LIN {X 0,Y 516.96,Z 356.095,A -85,B 0,C 180,E1 -5071.105,E2 -5071.105} C_VEL
LIN {X 0,Y 516.912,Z 356.1,A -85,B 0,C 180,E1 -5073.966,E2 -5073.966} C_VEL
LIN {X 0,Y 516.88,Z 356.104,A -85,B 0,C 180,E1 -5076.746,E2 -5076.746} C_VEL
LIN {X 0,Y 516.915,Z 356.098,A -85,B 0,C 180,E1 -5079.718,E2 -5079.718} C_VEL
LIN {X 0,Y 516.909,Z 356.099,A -85,B 0,C 180,E1 -5082.829,E2 -5082.829} C_VEL
LIN {X 0,Y 516.926,Z 356.097,A -85,B 0,C 180,E1 -5085.01,E2 -5085.01} C_VEL
LIN {X 0,Y 516.919,Z 356.099,A -85,B 0,C 180,E1 -5088.398,E2 -5088.398} C_VEL
LIN {X 0,Y 516.883,Z 356.103,A -85,B 0,C 180,E1 -5091.284,E2 -5091.284} C_VEL
LIN {X 0,Y 516.874,Z 356.103,A -85,B 0,C 180,E1 -5094.22,E2 -5094.22} C_VEL
LIN {X 0,Y 516.899,Z 356.103,A -85,B 0,C 180,E1 -5097.053,E2 -5097.053} C_VEL
LIN {X 0,Y 516.917,Z 356.245,A -85,B 0,C 180,E1 -5098.494,E2 -5098.494} C_VEL
LIN {X 0,Y 518.951,Z 365.114,A -85,B 0,C 180,E1 -5100.821,E2 -5100.821} C_VEL
LIN {X 0,Y 519.572,Z 369.036,A -85,B 0,C 180,E1 -5101.743,E2 -5101.743} C_VEL
LIN {X 0,Y 518.932,Z 379.362,A -85,B 0,C 180,E1 -5103.886,E2 -5103.886} C_VEL
LIN {X 0,Y 518.227,Z 395.981,A -85,B 0,C 180,E1 -5107.107,E2 -5107.107} C_VEL
LIN {X 0,Y 517.651,Z 412.713,A -85,B 0,C 180,E1 -5110.158,E2 -5110.158} C_VEL
LIN {X 0,Y 517.309,Z 428.9,A -85,B 0,C 180,E1 -5113.017,E2 -5113.017} C_VEL
LIN {X 0,Y 516.99,Z 447.206,A -85,B 0,C 180,E1 -5116.137,E2 -5116.137} C_VEL
LIN {X 0,Y 518.34,Z 458.651,A -85,B 0,C 180,E1 -5116.399,E2 -5116.399} C_VEL
LIN {X 0,Y 518.166,Z 471.053,A -85,B 0,C 180,E1 -5116.769,E2 -5116.769} C_VEL
LIN {X 0,Y 517.921,Z 483.766,A -85,B 0,C 180,E1 -5117.311,E2 -5117.311} C_VEL
LIN {X 0,Y 517.637,Z 495.546,A -85,B 0,C 180,E1 -5117.976,E2 -5117.976} C_VEL
LIN {X 0,Y 517.405,Z 506.176,A -85,B 0,C 180,E1 -5118.74,E2 -5118.74} C_VEL
LIN {X 0,Y 517.111,Z 516.148,A -85,B 0,C 180,E1 -5119.625,E2 -5119.625} C_VEL
LIN {X 0,Y 516.856,Z 525.214,A -85,B 0,C 180,E1 -5120.609,E2 -5120.609} C_VEL
LIN {X 0,Y 516.656,Z 534.061,A -85,B 0,C 180,E1 -5121.788,E2 -5121.788} C_VEL
LIN {X 0,Y 516.507,Z 541.106,A -85,B 0,C 180,E1 -5122.966,E2 -5122.966} C_VEL
LIN {X 0,Y 516.454,Z 546.751,A -85,B 0,C 180,E1 -5124.142,E2 -5124.142} C_VEL
LIN {X 0,Y 516.271,Z 551.161,A -85,B 0,C 180,E1 -5125.315,E2 -5125.315} C_VEL
LIN {X 0,Y 516.372,Z 553.512,A -85,B 0,C 180,E1 -5126.098,E2 -5126.098} C_VEL
LIN {X 0,Y 516.282,Z 555.403,A -85,B 0,C 180,E1 -5126.878,E2 -5126.878} C_VEL
LIN {X 0,Y 516.261,Z 556.824,A -85,B 0,C 180,E1 -5127.659,E2 -5127.659} C_VEL
LIN {X 0,Y 516.16,Z 558.448,A -85,B 0,C 180,E1 -5129.22,E2 -5129.22} C_VEL
LIN {X 0,Y 516.155,Z 558.67,A -85,B 0,C 180,E1 -5130,E2 -5130} C_VEL
LIN {X 0,Y 516.192,Z 557.838,A -85,B 0,C 180,E1 -5131.56,E2 -5131.56} C_VEL
LIN {X 0,Y 516.261,Z 556.835,A -85,B 0,C 180,E1 -5132.34,E2 -5132.34} C_VEL
LIN {X 0,Y 516.282,Z 555.417,A -85,B 0,C 180,E1 -5133.121,E2 -5133.121} C_VEL
LIN {X 0,Y 516.343,Z 552.441,A -85,B 0,C 180,E1 -5134.293,E2 -5134.293} C_VEL
LIN {X 0,Y 516.405,Z 548.405,A -85,B 0,C 180,E1 -5135.467,E2 -5135.467} C_VEL
LIN {X 0,Y 516.463,Z 543.024,A -85,B 0,C 180,E1 -5136.677,E2 -5136.677} C_VEL
LIN {X 0,Y 516.578,Z 536.641,A -85,B 0,C 180,E1 -5137.819,E2 -5137.819} C_VEL
LIN {X 0,Y 516.771,Z 528.471,A -85,B 0,C 180,E1 -5138.998,E2 -5138.998} C_VEL
LIN {X 0,Y 516.992,Z 520.13,A -85,B 0,C 180,E1 -5139.981,E2 -5139.981} C_VEL
LIN {X 0,Y 517.294,Z 509.933,A -85,B 0,C 180,E1 -5140.965,E2 -5140.965} C_VEL
LIN {X 0,Y 517.565,Z 498.759,A -85,B 0,C 180,E1 -5141.824,E2 -5141.824} C_VEL
LIN {X 0,Y 517.875,Z 486.984,A -85,B 0,C 180,E1 -5142.541,E2 -5142.541} C_VEL
LIN {X 0,Y 518.09,Z 475.398,A -85,B 0,C 180,E1 -5143.083,E2 -5143.083} C_VEL
LIN {X 0,Y 518.347,Z 462.076,A -85,B 0,C 180,E1 -5143.526,E2 -5143.526} C_VEL
LIN {X 0,Y 518.143,Z 456.418,A -85,B 0,C 180,E1 -5143.669,E2 -5143.669} C_VEL
LIN {X 0,Y 516.994,Z 447.607,A -85,B 0,C 180,E1 -5143.862,E2 -5143.862} C_VEL
LIN {X 0,Y 517.335,Z 430.732,A -85,B 0,C 180,E1 -5146.779,E2 -5146.779} C_VEL
LIN {X 0,Y 517.768,Z 411.104,A -85,B 0,C 180,E1 -5150.182,E2 -5150.182} C_VEL
LIN {X 0,Y 518.432,Z 392.937,A -85,B 0,C 180,E1 -5153.572,E2 -5153.572} C_VEL
LIN {X 0,Y 519.014,Z 377.127,A -85,B 0,C 180,E1 -5156.542,E2 -5156.542} C_VEL
LIN {X 0,Y 519.331,Z 367.451,A -85,B 0,C 180,E1 -5158.402,E2 -5158.402} C_VEL
LIN {X 0,Y 516.899,Z 356.101,A -85,B 0,C 180,E1 -5160.893,E2 -5160.893} C_VEL
LIN {X 0,Y 516.91,Z 356.098,A -85,B 0,C 180,E1 -5163.966,E2 -5163.966} C_VEL
LIN {X 0,Y 516.878,Z 356.103,A -85,B 0,C 180,E1 -5166.746,E2 -5166.746} C_VEL
LIN {X 0,Y 516.883,Z 356.099,A -85,B 0,C 180,E1 -5169.721,E2 -5169.721} C_VEL
LIN {X 0,Y 516.908,Z 356.095,A -85,B 0,C 180,E1 -5172.76,E2 -5172.76} C_VEL
LIN {X 0,Y 516.924,Z 356.097,A -85,B 0,C 180,E1 -5175.01,E2 -5175.01} C_VEL
LIN {X 0,Y 516.917,Z 356.099,A -85,B 0,C 180,E1 -5178.398,E2 -5178.398} C_VEL
LIN {X 0,Y 516.884,Z 356.098,A -85,B 0,C 180,E1 -5181.284,E2 -5181.284} C_VEL
LIN {X 0,Y 516.891,Z 356.098,A -85,B 0,C 180,E1 -5184.221,E2 -5184.221} C_VEL
LIN {X 0,Y 516.896,Z 356.1,A -85,B 0,C 180,E1 -5187.053,E2 -5187.053} C_VEL
LIN {X 0,Y 516.894,Z 356.098,A -85,B 0,C 180,E1 -5189.796,E2 -5189.796} C_VEL
LIN {X 0,Y 516.93,Z 356.092,A -85,B 0,C 180,E1 -5192.467,E2 -5192.467} C_VEL
LIN {X 0,Y 516.91,Z 356.098,A -85,B 0,C 180,E1 -5195.072,E2 -5195.072} C_VEL
LIN {X 0,Y 516.888,Z 356.102,A -85,B 0,C 180,E1 -5198.462,E2 -5198.462} C_VEL
LIN {X 0,Y 516.904,Z 356.095,A -85,B 0,C 180,E1 -5200.955,E2 -5200.955} C_VEL
LIN {X 0,Y 516.916,Z 356.097,A -85,B 0,C 180,E1 -5203.41,E2 -5203.41} C_VEL
LIN {X 0,Y 516.908,Z 356.096,A -85,B 0,C 180,E1 -5205.834,E2 -5205.834} C_VEL
LIN {X 0,Y 516.954,Z 356.091,A -85,B 0,C 180,E1 -5209.028,E2 -5209.028} C_VEL
LIN {X 0,Y 516.98,Z 356.088,A -85,B 0,C 180,E1 -5212.187,E2 -5212.187} C_VEL
LIN {X 0,Y 517.032,Z 356.079,A -85,B 0,C 180,E1 -5214.54,E2 -5214.54} C_VEL
LIN {X 0,Y 517.084,Z 356.074,A -85,B 0,C 180,E1 -5217.663,E2 -5217.663} C_VEL
LIN {X 0,Y 517.096,Z 356.073,A -85,B 0,C 180,E1 -5220.779,E2 -5220.779} C_VEL
LIN {X 0,Y 517.014,Z 356.083,A -85,B 0,C 180,E1 -5223.117,E2 -5223.117} C_VEL
LIN {X 0,Y 517.012,Z 356.082,A -85,B 0,C 180,E1 -5226.243,E2 -5226.243} C_VEL
LIN {X 0,Y 516.956,Z 356.09,A -85,B 0,C 180,E1 -5229.389,E2 -5229.389} C_VEL
LIN {X 0,Y 516.986,Z 356.09,A -85,B 0,C 180,E1 -5231.824,E2 -5231.824} C_VEL
LIN {X 0,Y 516.946,Z 356.094,A -85,B 0,C 180,E1 -5235.147,E2 -5235.147} C_VEL
LIN {X 0,Y 516.927,Z 356.094,A -85,B 0,C 180,E1 -5238.222,E2 -5238.222} C_VEL
LIN {X 0,Y 516.914,Z 356.096,A -85,B 0,C 180,E1 -5240.701,E2 -5240.701} C_VEL
LIN {X 0,Y 516.913,Z 356.095,A -85,B 0,C 180,E1 -5244.072,E2 -5244.072} C_VEL
LIN {X 0,Y 516.926,Z 356.094,A -85,B 0,C 180,E1 -5246.658,E2 -5246.658} C_VEL
LIN {X 0,Y 516.913,Z 356.095,A -85,B 0,C 180,E1 -5249.524,E2 -5249.524} C_VEL
LIN {X 0,Y 516.899,Z 356.097,A -85,B 0,C 180,E1 -5252.544,E2 -5252.544} C_VEL
LIN {X 0,Y 516.881,Z 356.103,A -85,B 0,C 180,E1 -5255.332,E2 -5255.332} C_VEL
LIN {X 0,Y 516.883,Z 356.097,A -85,B 0,C 180,E1 -5257.943,E2 -5257.943} C_VEL
LIN {X 0,Y 516.887,Z 356.1,A -85,B 0,C 180,E1 -5260.742,E2 -5260.742} C_VEL
LIN {X 0,Y 516.885,Z 356.098,A -85,B 0,C 180,E1 -5262.831,E2 -5262.831} C_VEL
LIN {X 0,Y 516.924,Z 356.096,A -85,B 0,C 180,E1 -5265.01,E2 -5265.01} C_VEL
LIN {X 0,Y 516.918,Z 356.096,A -85,B 0,C 180,E1 -5268.399,E2 -5268.399} C_VEL
LIN {X 0,Y 516.883,Z 356.102,A -85,B 0,C 180,E1 -5270.3,E2 -5270.3} C_VEL
LIN {X 0,Y 516.212,Z 356.183,A -85,B 0,C 180,E1 -5270.95,E2 -5270.95} C_VEL
LIN {X 0,Y 513.365,Z 356.541,A -85,B 0,C 180,E1 -5272.006,E2 -5272.006} C_VEL
LIN {X 0,Y 510.955,Z 356.843,A -85,B 0,C 180,E1 -5272.856,E2 -5272.856} C_VEL
LIN {X 0,Y 509.912,Z 356.971,A -85,B 0,C 180,E1 -5273.513,E2 -5273.513} C_VEL
LIN {X 0,Y 509.822,Z 356.98,A -85,B 0,C 180,E1 -5273.735,E2 -5273.735} C_VEL
LIN {X 0,Y 509.862,Z 356.974,A -85,B 0,C 180,E1 -5276.539,E2 -5276.539} C_VEL
LIN {X 0,Y 509.848,Z 356.973,A -85,B 0,C 180,E1 -5279.334,E2 -5279.334} C_VEL
LIN {X 0,Y 509.897,Z 356.973,A -85,B 0,C 180,E1 -5282.055,E2 -5282.055} C_VEL
LIN {X 0,Y 509.879,Z 356.972,A -85,B 0,C 180,E1 -5284.704,E2 -5284.704} C_VEL
LIN {X 0,Y 509.829,Z 356.978,A -85,B 0,C 180,E1 -5287.458,E2 -5287.458} C_VEL
LIN {X 0,Y 509.92,Z 356.966,A -85,B 0,C 180,E1 -5289.845,E2 -5289.845} C_VEL
LIN {X 0,Y 509.888,Z 356.97,A -85,B 0,C 180,E1 -5293.175,E2 -5293.175} C_VEL
LIN {X 0,Y 509.867,Z 356.976,A -85,B 0,C 180,E1 -5295.634,E2 -5295.634} C_VEL
LIN {X 0,Y 509.917,Z 356.969,A -85,B 0,C 180,E1 -5298.875,E2 -5298.875} C_VEL
LIN {X 0,Y 509.955,Z 356.967,A -85,B 0,C 180,E1 -5302.079,E2 -5302.079} C_VEL
LIN {X 0,Y 509.984,Z 356.958,A -85,B 0,C 180,E1 -5304.464,E2 -5304.464} C_VEL
LIN {X 0,Y 510.059,Z 356.949,A -85,B 0,C 180,E1 -5307.631,E2 -5307.631} C_VEL
LIN {X 0,Y 510.067,Z 356.949,A -85,B 0,C 180,E1 -5310.79,E2 -5310.79} C_VEL
LIN {X 0,Y 509.957,Z 356.96,A -85,B 0,C 180,E1 -5313.16,E2 -5313.16} C_VEL
LIN {X 0,Y 509.958,Z 356.961,A -85,B 0,C 180,E1 -5316.33,E2 -5316.33} C_VEL
LIN {X 0,Y 509.919,Z 356.969,A -85,B 0,C 180,E1 -5318.72,E2 -5318.72} C_VEL
LIN {X 0,Y 509.908,Z 356.971,A -85,B 0,C 180,E1 -5321.932,E2 -5321.932} C_VEL
LIN {X 0,Y 509.898,Z 356.971,A -85,B 0,C 180,E1 -5325.242,E2 -5325.242} C_VEL
LIN {X 0,Y 509.886,Z 356.97,A -85,B 0,C 180,E1 -5327.999,E2 -5327.999} C_VEL
LIN {X 0,Y 509.854,Z 356.975,A -85,B 0,C 180,E1 -5331.002,E2 -5331.002} C_VEL
LIN {X 0,Y 509.827,Z 356.981,A -85,B 0,C 180,E1 -5333.564,E2 -5333.564} C_VEL
LIN {X 0,Y 509.916,Z 356.966,A -85,B 0,C 180,E1 -5336.379,E2 -5336.379} C_VEL
LIN {X 0,Y 509.881,Z 356.975,A -85,B 0,C 180,E1 -5338.844,E2 -5338.844} C_VEL
LIN {X 0,Y 509.825,Z 356.979,A -85,B 0,C 180,E1 -5341.59,E2 -5341.59} C_VEL
LIN {X 0,Y 509.851,Z 356.974,A -85,B 0,C 180,E1 -5344.414,E2 -5344.414} C_VEL
LIN {X 0,Y 509.82,Z 356.982,A -85,B 0,C 180,E1 -5347.341,E2 -5347.341} C_VEL
LIN {X 0,Y 509.842,Z 356.979,A -85,B 0,C 180,E1 -5350.382,E2 -5350.382} C_VEL
LIN {X 0,Y 509.843,Z 356.976,A -85,B 0,C 180,E1 -5353.064,E2 -5353.064} C_VEL
LIN {X 0,Y 509.826,Z 356.979,A -85,B 0,C 180,E1 -5355.793,E2 -5355.793} C_VEL
LIN {X 0,Y 509.859,Z 356.975,A -85,B 0,C 180,E1 -5358.575,E2 -5358.575} C_VEL
LIN {X 0,Y 509.855,Z 356.976,A -85,B 0,C 180,E1 -5361.786,E2 -5361.786} C_VEL
LIN {X 0,Y 509.847,Z 356.975,A -85,B 0,C 180,E1 -5364.623,E2 -5364.623} C_VEL
LIN {X 0,Y 509.865,Z 356.975,A -85,B 0,C 180,E1 -5367.481,E2 -5367.481} C_VEL
LIN {X 0,Y 509.955,Z 357.04,A -85,B 0,C 180,E1 -5369.925,E2 -5369.925} C_VEL
LIN {X 0,Y 509.798,Z 363.427,A -85,B 0,C 180,E1 -5372.939,E2 -5372.939} C_VEL
LIN {X 0,Y 509.694,Z 369.046,A -85,B 0,C 180,E1 -5375.565,E2 -5375.565} C_VEL
LIN {X 0,Y 509.588,Z 374.525,A -85,B 0,C 180,E1 -5378.138,E2 -5378.138} C_VEL
LIN {X 0,Y 509.5,Z 379.893,A -85,B 0,C 180,E1 -5380.667,E2 -5380.667} C_VEL
LIN {X 0,Y 509.406,Z 385.315,A -85,B 0,C 180,E1 -5383.158,E2 -5383.158} C_VEL
LIN {X 0,Y 509.378,Z 390.782,A -85,B 0,C 180,E1 -5385.62,E2 -5385.62} C_VEL
LIN {X 0,Y 509.278,Z 398.149,A -85,B 0,C 180,E1 -5388.86,E2 -5388.86} C_VEL
LIN {X 0,Y 509.269,Z 404.776,A -85,B 0,C 180,E1 -5391.718,E2 -5391.718} C_VEL
LIN {X 0,Y 510.102,Z 412.51,A -85,B 0,C 180,E1 -5392.031,E2 -5392.031} C_VEL
LIN {X 0,Y 509.994,Z 422.565,A -85,B 0,C 180,E1 -5392.577,E2 -5392.577} C_VEL
LIN {X 0,Y 509.86,Z 430.431,A -85,B 0,C 180,E1 -5393.156,E2 -5393.156} C_VEL
LIN {X 0,Y 509.631,Z 437.924,A -85,B 0,C 180,E1 -5393.865,E2 -5393.865} C_VEL
LIN {X 0,Y 509.591,Z 444.394,A -85,B 0,C 180,E1 -5394.658,E2 -5394.658} C_VEL
LIN {X 0,Y 509.512,Z 450.616,A -85,B 0,C 180,E1 -5395.649,E2 -5395.649} C_VEL
LIN {X 0,Y 509.513,Z 454.382,A -85,B 0,C 180,E1 -5396.441,E2 -5396.441} C_VEL
LIN {X 0,Y 509.254,Z 458.441,A -85,B 0,C 180,E1 -5397.627,E2 -5397.627} C_VEL
LIN {X 0,Y 509.191,Z 460.209,A -85,B 0,C 180,E1 -5398.418,E2 -5398.418} C_VEL
LIN {X 0,Y 509.173,Z 461.279,A -85,B 0,C 180,E1 -5399.209,E2 -5399.209} C_VEL
LIN {X 0,Y 509.173,Z 461.683,A -85,B 0,C 180,E1 -5400,E2 -5400} C_VEL
LIN {X 0,Y 509.179,Z 461.428,A -85,B 0,C 180,E1 -5400.791,E2 -5400.791} C_VEL
LIN {X 0,Y 509.202,Z 460.51,A -85,B 0,C 180,E1 -5401.582,E2 -5401.582} C_VEL
LIN {X 0,Y 509.381,Z 457.808,A -85,B 0,C 180,E1 -5402.768,E2 -5402.768} C_VEL
LIN {X 0,Y 509.51,Z 455.083,A -85,B 0,C 180,E1 -5403.559,E2 -5403.559} C_VEL
LIN {X 0,Y 509.532,Z 450.473,A -85,B 0,C 180,E1 -5404.549,E2 -5404.549} C_VEL
LIN {X 0,Y 509.641,Z 445.61,A -85,B 0,C 180,E1 -5405.341,E2 -5405.341} C_VEL
LIN {X 0,Y 509.731,Z 439.426,A -85,B 0,C 180,E1 -5406.134,E2 -5406.134} C_VEL
LIN {X 0,Y 509.963,Z 432.423,A -85,B 0,C 180,E1 -5406.838,E2 -5406.838} C_VEL
LIN {X 0,Y 510.044,Z 424.158,A -85,B 0,C 180,E1 -5407.482,E2 -5407.482} C_VEL
LIN {X 0,Y 510.246,Z 414.949,A -85,B 0,C 180,E1 -5408.017,E2 -5408.017} C_VEL
LIN {X 0,Y 509.775,Z 408.095,A -85,B 0,C 180,E1 -5408.323,E2 -5408.323} C_VEL
LIN {X 0,Y 509.349,Z 405.631,A -85,B 0,C 180,E1 -5408.43,E2 -5408.43} C_VEL
LIN {X 0,Y 509.46,Z 398.545,A -85,B 0,C 180,E1 -5411.636,E2 -5411.636} C_VEL
LIN {X 0,Y 509.576,Z 390.773,A -85,B 0,C 180,E1 -5415.192,E2 -5415.192} C_VEL
LIN {X 0,Y 509.663,Z 383.695,A -85,B 0,C 180,E1 -5418.491,E2 -5418.491} C_VEL
LIN {X 0,Y 509.766,Z 378.33,A -85,B 0,C 180,E1 -5421.005,E2 -5421.005} C_VEL
LIN {X 0,Y 509.885,Z 372.925,A -85,B 0,C 180,E1 -5423.561,E2 -5423.561} C_VEL
LIN {X 0,Y 510.067,Z 367.004,A -85,B 0,C 180,E1 -5426.413,E2 -5426.413} C_VEL
LIN {X 0,Y 510.222,Z 360.055,A -85,B 0,C 180,E1 -5429.728,E2 -5429.728} C_VEL
LIN {X 0,Y 509.89,Z 356.976,A -85,B 0,C 180,E1 -5431.287,E2 -5431.287} C_VEL
LIN {X 0,Y 509.851,Z 356.979,A -85,B 0,C 180,E1 -5434.414,E2 -5434.414} C_VEL
LIN {X 0,Y 509.82,Z 356.982,A -85,B 0,C 180,E1 -5437.341,E2 -5437.341} C_VEL
LIN {X 0,Y 509.866,Z 356.977,A -85,B 0,C 180,E1 -5440.38,E2 -5440.38} C_VEL
LIN {X 0,Y 509.844,Z 356.98,A -85,B 0,C 180,E1 -5443.064,E2 -5443.064} C_VEL
LIN {X 0,Y 509.834,Z 356.98,A -85,B 0,C 180,E1 -5445.792,E2 -5445.792} C_VEL
LIN {X 0,Y 509.861,Z 356.978,A -85,B 0,C 180,E1 -5448.575,E2 -5448.575} C_VEL
LIN {X 0,Y 509.853,Z 356.979,A -85,B 0,C 180,E1 -5451.786,E2 -5451.786} C_VEL
LIN {X 0,Y 509.833,Z 356.982,A -85,B 0,C 180,E1 -5454.622,E2 -5454.622} C_VEL
LIN {X 0,Y 509.867,Z 356.979,A -85,B 0,C 180,E1 -5457.481,E2 -5457.481} C_VEL
LIN {X 0,Y 509.874,Z 357.195,A -85,B 0,C 180,E1 -5458.065,E2 -5458.065} C_VEL
LIN {X 0,Y 511.829,Z 365.557,A -85,B 0,C 180,E1 -5460.375,E2 -5460.375} C_VEL
LIN {X 0,Y 512.613,Z 369.385,A -85,B 0,C 180,E1 -5461.336,E2 -5461.336} C_VEL
LIN {X 0,Y 512.479,Z 375.336,A -85,B 0,C 180,E1 -5462.651,E2 -5462.651} C_VEL
LIN {X 0,Y 511.447,Z 391.148,A -85,B 0,C 180,E1 -5465.87,E2 -5465.87} C_VEL
LIN {X 0,Y 510.911,Z 404.42,A -85,B 0,C 180,E1 -5468.409,E2 -5468.409} C_VEL
LIN {X 0,Y 510.48,Z 420.361,A -85,B 0,C 180,E1 -5471.331,E2 -5471.331} C_VEL
LIN {X 0,Y 510.135,Z 434.33,A -85,B 0,C 180,E1 -5473.801,E2 -5473.801} C_VEL
LIN {X 0,Y 509.904,Z 446.963,A -85,B 0,C 180,E1 -5476.004,E2 -5476.004} C_VEL
LIN {X 0,Y 511.335,Z 459.512,A -85,B 0,C 180,E1 -5476.285,E2 -5476.285} C_VEL
LIN {X 0,Y 511.157,Z 472.121,A -85,B 0,C 180,E1 -5476.685,E2 -5476.685} C_VEL
LIN {X 0,Y 510.896,Z 483.442,A -85,B 0,C 180,E1 -5477.184,E2 -5477.184} C_VEL
LIN {X 0,Y 510.59,Z 495.851,A -85,B 0,C 180,E1 -5477.903,E2 -5477.903} C_VEL
LIN {X 0,Y 510.275,Z 507.551,A -85,B 0,C 180,E1 -5478.782,E2 -5478.782} C_VEL
LIN {X 0,Y 510.011,Z 517.204,A -85,B 0,C 180,E1 -5479.68,E2 -5479.68} C_VEL
LIN {X 0,Y 509.759,Z 526,A -85,B 0,C 180,E1 -5480.677,E2 -5480.677} C_VEL
LIN {X 0,Y 509.563,Z 534.517,A -85,B 0,C 180,E1 -5481.873,E2 -5481.873} C_VEL
LIN {X 0,Y 509.401,Z 541.831,A -85,B 0,C 180,E1 -5483.155,E2 -5483.155} C_VEL
LIN {X 0,Y 509.344,Z 547.652,A -85,B 0,C 180,E1 -5484.457,E2 -5484.457} C_VEL
LIN {X 0,Y 509.268,Z 551.717,A -85,B 0,C 180,E1 -5485.647,E2 -5485.647} C_VEL
LIN {X 0,Y 509.232,Z 554.719,A -85,B 0,C 180,E1 -5486.835,E2 -5486.835} C_VEL
LIN {X 0,Y 509.19,Z 556.147,A -85,B 0,C 180,E1 -5487.627,E2 -5487.627} C_VEL
LIN {X 0,Y 509.091,Z 557.783,A -85,B 0,C 180,E1 -5489.209,E2 -5489.209} C_VEL
LIN {X 0,Y 509.086,Z 558.011,A -85,B 0,C 180,E1 -5490,E2 -5490} C_VEL
LIN {X 0,Y 509.09,Z 557.794,A -85,B 0,C 180,E1 -5490.791,E2 -5490.791} C_VEL
LIN {X 0,Y 509.19,Z 556.177,A -85,B 0,C 180,E1 -5492.373,E2 -5492.373} C_VEL
LIN {X 0,Y 509.232,Z 554.758,A -85,B 0,C 180,E1 -5493.164,E2 -5493.164} C_VEL
LIN {X 0,Y 509.268,Z 551.773,A -85,B 0,C 180,E1 -5494.353,E2 -5494.353} C_VEL
LIN {X 0,Y 509.344,Z 547.726,A -85,B 0,C 180,E1 -5495.543,E2 -5495.543} C_VEL
LIN {X 0,Y 509.401,Z 541.937,A -85,B 0,C 180,E1 -5496.844,E2 -5496.844} C_VEL
LIN {X 0,Y 509.538,Z 534.659,A -85,B 0,C 180,E1 -5498.127,E2 -5498.127} C_VEL
LIN {X 0,Y 509.759,Z 526.19,A -85,B 0,C 180,E1 -5499.323,E2 -5499.323} C_VEL
LIN {X 0,Y 510.007,Z 517.446,A -85,B 0,C 180,E1 -5500.32,E2 -5500.32} C_VEL
LIN {X 0,Y 510.336,Z 506.668,A -85,B 0,C 180,E1 -5501.317,E2 -5501.317} C_VEL
LIN {X 0,Y 510.591,Z 496.03,A -85,B 0,C 180,E1 -5502.111,E2 -5502.111} C_VEL
LIN {X 0,Y 510.927,Z 483.941,A -85,B 0,C 180,E1 -5502.815,E2 -5502.815} C_VEL
LIN {X 0,Y 511.177,Z 471.424,A -85,B 0,C 180,E1 -5503.365,E2 -5503.365} C_VEL
LIN {X 0,Y 511.344,Z 458.446,A -85,B 0,C 180,E1 -5503.765,E2 -5503.765} C_VEL
LIN {X 0,Y 509.915,Z 447.23,A -85,B 0,C 180,E1 -5504.033,E2 -5504.033} C_VEL
LIN {X 0,Y 510.234,Z 433.939,A -85,B 0,C 180,E1 -5506.401,E2 -5506.401} C_VEL
LIN {X 0,Y 510.662,Z 416.277,A -85,B 0,C 180,E1 -5509.496,E2 -5509.496} C_VEL
LIN {X 0,Y 511.084,Z 402.777,A -85,B 0,C 180,E1 -5512.007,E2 -5512.007} C_VEL
LIN {X 0,Y 511.662,Z 388.832,A -85,B 0,C 180,E1 -5514.665,E2 -5514.665} C_VEL
LIN {X 0,Y 512.427,Z 372.555,A -85,B 0,C 180,E1 -5517.795,E2 -5517.795} C_VEL
LIN {X 0,Y 512.349,Z 368.581,A -85,B 0,C 180,E1 -5518.609,E2 -5518.609} C_VEL
LIN {X 0,Y 509.847,Z 356.979,A -85,B 0,C 180,E1 -5521.206,E2 -5521.206} C_VEL
LIN {X 0,Y 509.858,Z 356.975,A -85,B 0,C 180,E1 -5524.202,E2 -5524.202} C_VEL
LIN {X 0,Y 509.818,Z 356.979,A -85,B 0,C 180,E1 -5527.341,E2 -5527.341} C_VEL
LIN {X 0,Y 509.84,Z 356.979,A -85,B 0,C 180,E1 -5530.382,E2 -5530.382} C_VEL
LIN {X 0,Y 509.842,Z 356.977,A -85,B 0,C 180,E1 -5533.064,E2 -5533.064} C_VEL
LIN {X 0,Y 509.832,Z 356.977,A -85,B 0,C 180,E1 -5535.792,E2 -5535.792} C_VEL
LIN {X 0,Y 509.858,Z 356.977,A -85,B 0,C 180,E1 -5538.575,E2 -5538.575} C_VEL
LIN {X 0,Y 509.854,Z 356.978,A -85,B 0,C 180,E1 -5541.786,E2 -5541.786} C_VEL
LIN {X 0,Y 509.845,Z 356.976,A -85,B 0,C 180,E1 -5544.623,E2 -5544.623} C_VEL
LIN {X 0,Y 509.863,Z 356.973,A -85,B 0,C 180,E1 -5547.481,E2 -5547.481} C_VEL
LIN {X 0,Y 509.86,Z 356.977,A -85,B 0,C 180,E1 -5550.274,E2 -5550.274} C_VEL
LIN {X 0,Y 509.887,Z 356.97,A -85,B 0,C 180,E1 -5552.944,E2 -5552.944} C_VEL
LIN {X 0,Y 509.865,Z 356.975,A -85,B 0,C 180,E1 -5555.574,E2 -5555.574} C_VEL
LIN {X 0,Y 509.852,Z 356.976,A -85,B 0,C 180,E1 -5558.998,E2 -5558.998} C_VEL
LIN {X 0,Y 509.89,Z 356.973,A -85,B 0,C 180,E1 -5561.999,E2 -5561.999} C_VEL
LIN {X 0,Y 509.912,Z 356.968,A -85,B 0,C 180,E1 -5564.819,E2 -5564.819} C_VEL
LIN {X 0,Y 509.903,Z 356.97,A -85,B 0,C 180,E1 -5568.124,E2 -5568.124} C_VEL
LIN {X 0,Y 509.917,Z 356.966,A -85,B 0,C 180,E1 -5571.28,E2 -5571.28} C_VEL
LIN {X 0,Y 509.98,Z 356.963,A -85,B 0,C 180,E1 -5573.67,E2 -5573.67} C_VEL
LIN {X 0,Y 510.056,Z 356.949,A -85,B 0,C 180,E1 -5577.631,E2 -5577.631} C_VEL
LIN {X 0,Y 510.066,Z 356.948,A -85,B 0,C 180,E1 -5580.789,E2 -5580.789} C_VEL
LIN {X 0,Y 509.956,Z 356.962,A -85,B 0,C 180,E1 -5583.16,E2 -5583.16} C_VEL
LIN {X 0,Y 509.98,Z 356.958,A -85,B 0,C 180,E1 -5586.33,E2 -5586.33} C_VEL
LIN {X 0,Y 509.918,Z 356.97,A -85,B 0,C 180,E1 -5588.72,E2 -5588.72} C_VEL
LIN {X 0,Y 509.953,Z 356.965,A -85,B 0,C 180,E1 -5591.931,E2 -5591.931} C_VEL
LIN {X 0,Y 509.895,Z 356.974,A -85,B 0,C 180,E1 -5595.242,E2 -5595.242} C_VEL
LIN {X 0,Y 509.89,Z 356.97,A -85,B 0,C 180,E1 -5598.001,E2 -5598.001} C_VEL
LIN {X 0,Y 509.852,Z 356.975,A -85,B 0,C 180,E1 -5601.002,E2 -5601.002} C_VEL
LIN {X 0,Y 509.839,Z 356.98,A -85,B 0,C 180,E1 -5603.563,E2 -5603.563} C_VEL
LIN {X 0,Y 509.913,Z 356.966,A -85,B 0,C 180,E1 -5606.379,E2 -5606.379} C_VEL
LIN {X 0,Y 509.878,Z 356.975,A -85,B 0,C 180,E1 -5608.844,E2 -5608.844} C_VEL
LIN {X 0,Y 509.823,Z 356.98,A -85,B 0,C 180,E1 -5611.59,E2 -5611.59} C_VEL
LIN {X 0,Y 509.854,Z 356.974,A -85,B 0,C 180,E1 -5614.413,E2 -5614.413} C_VEL
LIN {X 0,Y 509.82,Z 356.979,A -85,B 0,C 180,E1 -5617.341,E2 -5617.341} C_VEL
LIN {X 0,Y 509.84,Z 356.98,A -85,B 0,C 180,E1 -5620.382,E2 -5620.382} C_VEL
LIN {X 0,Y 509.825,Z 356.978,A -85,B 0,C 180,E1 -5623.062,E2 -5623.062} C_VEL
LIN {X 0,Y 509.833,Z 356.978,A -85,B 0,C 180,E1 -5625.792,E2 -5625.792} C_VEL
LIN {X 0,Y 509.859,Z 356.977,A -85,B 0,C 180,E1 -5628.575,E2 -5628.575} C_VEL
LIN {X 0,Y 509.853,Z 356.977,A -85,B 0,C 180,E1 -5631.787,E2 -5631.787} C_VEL
LIN {X 0,Y 509.822,Z 356.98,A -85,B 0,C 180,E1 -5633.735,E2 -5633.735} C_VEL
LIN {X 0,Y 509.154,Z 357.062,A -85,B 0,C 180,E1 -5634.395,E2 -5634.395} C_VEL
LIN {X 0,Y 506.342,Z 357.415,A -85,B 0,C 180,E1 -5635.467,E2 -5635.467} C_VEL
LIN {X 0,Y 503.955,Z 357.714,A -85,B 0,C 180,E1 -5636.331,E2 -5636.331} C_VEL
LIN {X 0,Y 502.908,Z 357.843,A -85,B 0,C 180,E1 -5636.997,E2 -5636.997} C_VEL
LIN {X 0,Y 502.811,Z 357.853,A -85,B 0,C 180,E1 -5637.223,E2 -5637.223} C_VEL
LIN {X 0,Y 502.817,Z 357.852,A -85,B 0,C 180,E1 -5640.065,E2 -5640.065} C_VEL
LIN {X 0,Y 502.837,Z 357.849,A -85,B 0,C 180,E1 -5642.534,E2 -5642.534} C_VEL
LIN {X 0,Y 502.829,Z 357.852,A -85,B 0,C 180,E1 -5645.299,E2 -5645.299} C_VEL
LIN {X 0,Y 502.783,Z 357.855,A -85,B 0,C 180,E1 -5647.827,E2 -5647.827} C_VEL
LIN {X 0,Y 502.829,Z 357.854,A -85,B 0,C 180,E1 -5650.4,E2 -5650.4} C_VEL
LIN {X 0,Y 502.838,Z 357.848,A -85,B 0,C 180,E1 -5652.932,E2 -5652.932} C_VEL
LIN {X 0,Y 502.848,Z 357.85,A -85,B 0,C 180,E1 -5655.429,E2 -5655.429} C_VEL
LIN {X 0,Y 502.881,Z 357.846,A -85,B 0,C 180,E1 -5658.717,E2 -5658.717} C_VEL
LIN {X 0,Y 502.905,Z 357.844,A -85,B 0,C 180,E1 -5661.967,E2 -5661.967} C_VEL
LIN {X 0,Y 502.938,Z 357.836,A -85,B 0,C 180,E1 -5664.387,E2 -5664.387} C_VEL
LIN {X 0,Y 503.028,Z 357.826,A -85,B 0,C 180,E1 -5667.598,E2 -5667.598} C_VEL
LIN {X 0,Y 503.031,Z 357.826,A -85,B 0,C 180,E1 -5670,E2 -5670} C_VEL
LIN {X 0,Y 503.028,Z 357.825,A -85,B 0,C 180,E1 -5672.402,E2 -5672.402} C_VEL
LIN {X 0,Y 502.937,Z 357.84,A -85,B 0,C 180,E1 -5675.614,E2 -5675.614} C_VEL
LIN {X 0,Y 502.906,Z 357.84,A -85,B 0,C 180,E1 -5678.033,E2 -5678.033} C_VEL
LIN {X 0,Y 502.882,Z 357.842,A -85,B 0,C 180,E1 -5681.283,E2 -5681.283} C_VEL
LIN {X 0,Y 502.849,Z 357.846,A -85,B 0,C 180,E1 -5684.571,E2 -5684.571} C_VEL
LIN {X 0,Y 502.859,Z 357.846,A -85,B 0,C 180,E1 -5687.907,E2 -5687.907} C_VEL
LIN {X 0,Y 502.832,Z 357.852,A -85,B 0,C 180,E1 -5690.536,E2 -5690.536} C_VEL
LIN {X 0,Y 502.792,Z 357.853,A -85,B 0,C 180,E1 -5693.041,E2 -5693.041} C_VEL
LIN {X 0,Y 502.826,Z 357.852,A -85,B 0,C 180,E1 -5695.677,E2 -5695.677} C_VEL
LIN {X 0,Y 502.844,Z 357.849,A -85,B 0,C 180,E1 -5698.373,E2 -5698.373} C_VEL
LIN {X 0,Y 502.797,Z 357.854,A -85,B 0,C 180,E1 -5701.499,E2 -5701.499} C_VEL
LIN {X 0,Y 502.807,Z 357.854,A -85,B 0,C 180,E1 -5703.994,E2 -5703.994} C_VEL
LIN {X 0,Y 502.781,Z 357.86,A -85,B 0,C 180,E1 -5707.178,E2 -5707.178} C_VEL
LIN {X 0,Y 502.791,Z 357.855,A -85,B 0,C 180,E1 -5710.015,E2 -5710.015} C_VEL
LIN {X 0,Y 502.806,Z 357.855,A -85,B 0,C 180,E1 -5712.199,E2 -5712.199} C_VEL
LIN {X 0,Y 502.789,Z 357.859,A -85,B 0,C 180,E1 -5715.47,E2 -5715.47} C_VEL
LIN {X 0,Y 502.823,Z 357.855,A -85,B 0,C 180,E1 -5718.934,E2 -5718.934} C_VEL
LIN {X 0,Y 502.798,Z 357.856,A -85,B 0,C 180,E1 -5722.046,E2 -5722.046} C_VEL
LIN {X 0,Y 502.811,Z 357.853,A -85,B 0,C 180,E1 -5725.035,E2 -5725.035} C_VEL
LIN {X 0,Y 502.788,Z 357.854,A -85,B 0,C 180,E1 -5727.916,E2 -5727.916} C_VEL
LIN {X 0,Y 502.916,Z 357.909,A -85,B 0,C 180,E1 -5729.875,E2 -5729.875} C_VEL
LIN {X 0,Y 502.762,Z 363.466,A -85,B 0,C 180,E1 -5732.529,E2 -5732.529} C_VEL
LIN {X 0,Y 502.663,Z 369.435,A -85,B 0,C 180,E1 -5735.341,E2 -5735.341} C_VEL
LIN {X 0,Y 502.574,Z 374.743,A -85,B 0,C 180,E1 -5737.817,E2 -5737.817} C_VEL
LIN {X 0,Y 502.466,Z 380.261,A -85,B 0,C 180,E1 -5740.386,E2 -5740.386} C_VEL
LIN {X 0,Y 502.367,Z 385.678,A -85,B 0,C 180,E1 -5742.915,E2 -5742.915} C_VEL
LIN {X 0,Y 502.353,Z 391.14,A -85,B 0,C 180,E1 -5745.415,E2 -5745.415} C_VEL
LIN {X 0,Y 502.236,Z 398.504,A -85,B 0,C 180,E1 -5748.702,E2 -5748.702} C_VEL
LIN {X 0,Y 502.212,Z 405.071,A -85,B 0,C 180,E1 -5751.576,E2 -5751.576} C_VEL
LIN {X 0,Y 503.117,Z 413.314,A -85,B 0,C 180,E1 -5751.92,E2 -5751.92} C_VEL
LIN {X 0,Y 503.008,Z 423.248,A -85,B 0,C 180,E1 -5752.473,E2 -5752.473} C_VEL
LIN {X 0,Y 502.84,Z 431.409,A -85,B 0,C 180,E1 -5753.089,E2 -5753.089} C_VEL
LIN {X 0,Y 502.599,Z 438.532,A -85,B 0,C 180,E1 -5753.779,E2 -5753.779} C_VEL
LIN {X 0,Y 502.563,Z 445.009,A -85,B 0,C 180,E1 -5754.584,E2 -5754.584} C_VEL
LIN {X 0,Y 502.48,Z 451.23,A -85,B 0,C 180,E1 -5755.588,E2 -5755.588} C_VEL
LIN {X 0,Y 502.466,Z 455.006,A -85,B 0,C 180,E1 -5756.391,E2 -5756.391} C_VEL
LIN {X 0,Y 502.336,Z 457.929,A -85,B 0,C 180,E1 -5757.193,E2 -5757.193} C_VEL
LIN {X 0,Y 502.125,Z 460.869,A -85,B 0,C 180,E1 -5758.396,E2 -5758.396} C_VEL
LIN {X 0,Y 502.106,Z 461.949,A -85,B 0,C 180,E1 -5759.198,E2 -5759.198} C_VEL
LIN {X 0,Y 502.106,Z 462.361,A -85,B 0,C 180,E1 -5760,E2 -5760} C_VEL
LIN {X 0,Y 502.113,Z 462.114,A -85,B 0,C 180,E1 -5760.802,E2 -5760.802} C_VEL
LIN {X 0,Y 502.14,Z 461.202,A -85,B 0,C 180,E1 -5761.604,E2 -5761.604} C_VEL
LIN {X 0,Y 502.339,Z 458.513,A -85,B 0,C 180,E1 -5762.807,E2 -5762.807} C_VEL
LIN {X 0,Y 502.477,Z 455.786,A -85,B 0,C 180,E1 -5763.609,E2 -5763.609} C_VEL
LIN {X 0,Y 502.503,Z 451.187,A -85,B 0,C 180,E1 -5764.613,E2 -5764.613} C_VEL
LIN {X 0,Y 502.627,Z 446.34,A -85,B 0,C 180,E1 -5765.416,E2 -5765.416} C_VEL
LIN {X 0,Y 502.728,Z 440.183,A -85,B 0,C 180,E1 -5766.22,E2 -5766.22} C_VEL
LIN {X 0,Y 502.942,Z 433.408,A -85,B 0,C 180,E1 -5766.918,E2 -5766.918} C_VEL
LIN {X 0,Y 503.072,Z 425.075,A -85,B 0,C 180,E1 -5767.586,E2 -5767.586} C_VEL
LIN {X 0,Y 503.274,Z 416.035,A -85,B 0,C 180,E1 -5768.128,E2 -5768.128} C_VEL
LIN {X 0,Y 502.889,Z 409.413,A -85,B 0,C 180,E1 -5768.438,E2 -5768.438} C_VEL
LIN {X 0,Y 502.325,Z 406.05,A -85,B 0,C 180,E1 -5768.6,E2 -5768.6} C_VEL
LIN {X 0,Y 502.42,Z 399.224,A -85,B 0,C 180,E1 -5771.71,E2 -5771.71} C_VEL
LIN {X 0,Y 502.538,Z 391.237,A -85,B 0,C 180,E1 -5775.41,E2 -5775.41} C_VEL
LIN {X 0,Y 502.634,Z 385.624,A -85,B 0,C 180,E1 -5778.047,E2 -5778.047} C_VEL
LIN {X 0,Y 502.775,Z 378.76,A -85,B 0,C 180,E1 -5781.312,E2 -5781.312} C_VEL
LIN {X 0,Y 502.906,Z 373.397,A -85,B 0,C 180,E1 -5783.908,E2 -5783.908} C_VEL
LIN {X 0,Y 503.064,Z 367.79,A -85,B 0,C 180,E1 -5786.606,E2 -5786.606} C_VEL
LIN {X 0,Y 503.207,Z 362.373,A -85,B 0,C 180,E1 -5789.263,E2 -5789.263} C_VEL
LIN {X 0,Y 503.002,Z 358.693,A -85,B 0,C 180,E1 -5791.129,E2 -5791.129} C_VEL
LIN {X 0,Y 502.815,Z 357.857,A -85,B 0,C 180,E1 -5791.595,E2 -5791.595} C_VEL
LIN {X 0,Y 502.803,Z 357.858,A -85,B 0,C 180,E1 -5794.443,E2 -5794.443} C_VEL
LIN {X 0,Y 502.781,Z 357.859,A -85,B 0,C 180,E1 -5797.178,E2 -5797.178} C_VEL
LIN {X 0,Y 502.83,Z 357.854,A -85,B 0,C 180,E1 -5800.011,E2 -5800.011} C_VEL
LIN {X 0,Y 502.827,Z 357.854,A -85,B 0,C 180,E1 -5802.202,E2 -5802.202} C_VEL
LIN {X 0,Y 502.804,Z 357.857,A -85,B 0,C 180,E1 -5805.468,E2 -5805.468} C_VEL
LIN {X 0,Y 502.833,Z 357.853,A -85,B 0,C 180,E1 -5807.864,E2 -5807.864} C_VEL
LIN {X 0,Y 502.804,Z 357.856,A -85,B 0,C 180,E1 -5811.024,E2 -5811.024} C_VEL
LIN {X 0,Y 502.778,Z 357.859,A -85,B 0,C 180,E1 -5814.169,E2 -5814.169} C_VEL
LIN {X 0,Y 502.846,Z 357.854,A -85,B 0,C 180,E1 -5817.446,E2 -5817.446} C_VEL
LIN {X 0,Y 503.131,Z 359.181,A -85,B 0,C 180,E1 -5817.94,E2 -5817.94} C_VEL
LIN {X 0,Y 505.098,Z 367.869,A -85,B 0,C 180,E1 -5820.399,E2 -5820.399} C_VEL
LIN {X 0,Y 505.847,Z 372.11,A -85,B 0,C 180,E1 -5821.47,E2 -5821.47} C_VEL
LIN {X 0,Y 505.355,Z 379.995,A -85,B 0,C 180,E1 -5823.207,E2 -5823.207} C_VEL
LIN {X 0,Y 504.395,Z 395.332,A -85,B 0,C 180,E1 -5826.38,E2 -5826.38} C_VEL
LIN {X 0,Y 503.714,Z 412.011,A -85,B 0,C 180,E1 -5829.585,E2 -5829.585} C_VEL
LIN {X 0,Y 503.251,Z 429.137,A -85,B 0,C 180,E1 -5832.737,E2 -5832.737} C_VEL
LIN {X 0,Y 502.849,Z 446.578,A -85,B 0,C 180,E1 -5835.842,E2 -5835.842} C_VEL
LIN {X 0,Y 504.336,Z 460.292,A -85,B 0,C 180,E1 -5836.168,E2 -5836.168} C_VEL
LIN {X 0,Y 504.128,Z 473.162,A -85,B 0,C 180,E1 -5836.599,E2 -5836.599} C_VEL
LIN {X 0,Y 503.871,Z 484.124,A -85,B 0,C 180,E1 -5837.105,E2 -5837.105} C_VEL
LIN {X 0,Y 503.547,Z 496.101,A -85,B 0,C 180,E1 -5837.827,E2 -5837.827} C_VEL
LIN {X 0,Y 503.2,Z 507.738,A -85,B 0,C 180,E1 -5838.724,E2 -5838.724} C_VEL
LIN {X 0,Y 502.956,Z 516.272,A -85,B 0,C 180,E1 -5839.534,E2 -5839.534} C_VEL
LIN {X 0,Y 502.708,Z 525.136,A -85,B 0,C 180,E1 -5840.545,E2 -5840.545} C_VEL
LIN {X 0,Y 502.495,Z 533.714,A -85,B 0,C 180,E1 -5841.758,E2 -5841.758} C_VEL
LIN {X 0,Y 502.332,Z 540.705,A -85,B 0,C 180,E1 -5842.988,E2 -5842.988} C_VEL
LIN {X 0,Y 502.282,Z 546.926,A -85,B 0,C 180,E1 -5844.379,E2 -5844.379} C_VEL
LIN {X 0,Y 502.178,Z 551.012,A -85,B 0,C 180,E1 -5845.585,E2 -5845.585} C_VEL
LIN {X 0,Y 502.182,Z 554.034,A -85,B 0,C 180,E1 -5846.791,E2 -5846.791} C_VEL
LIN {X 0,Y 502.122,Z 555.471,A -85,B 0,C 180,E1 -5847.593,E2 -5847.593} C_VEL
LIN {X 0,Y 502.021,Z 557.12,A -85,B 0,C 180,E1 -5849.198,E2 -5849.198} C_VEL
LIN {X 0,Y 502.017,Z 557.351,A -85,B 0,C 180,E1 -5850,E2 -5850} C_VEL
LIN {X 0,Y 502.02,Z 557.136,A -85,B 0,C 180,E1 -5850.802,E2 -5850.802} C_VEL
LIN {X 0,Y 502.122,Z 555.521,A -85,B 0,C 180,E1 -5852.406,E2 -5852.406} C_VEL
LIN {X 0,Y 502.182,Z 554.098,A -85,B 0,C 180,E1 -5853.209,E2 -5853.209} C_VEL
LIN {X 0,Y 502.178,Z 551.103,A -85,B 0,C 180,E1 -5854.414,E2 -5854.414} C_VEL
LIN {X 0,Y 502.281,Z 547.046,A -85,B 0,C 180,E1 -5855.621,E2 -5855.621} C_VEL
LIN {X 0,Y 502.332,Z 540.873,A -85,B 0,C 180,E1 -5857.011,E2 -5857.011} C_VEL
LIN {X 0,Y 502.483,Z 533.93,A -85,B 0,C 180,E1 -5858.242,E2 -5858.242} C_VEL
LIN {X 0,Y 502.708,Z 525.413,A -85,B 0,C 180,E1 -5859.455,E2 -5859.455} C_VEL
LIN {X 0,Y 502.98,Z 516.618,A -85,B 0,C 180,E1 -5860.465,E2 -5860.465} C_VEL
LIN {X 0,Y 503.346,Z 505.787,A -85,B 0,C 180,E1 -5861.476,E2 -5861.476} C_VEL
LIN {X 0,Y 503.595,Z 495.331,A -85,B 0,C 180,E1 -5862.263,E2 -5862.263} C_VEL
LIN {X 0,Y 503.903,Z 483.786,A -85,B 0,C 180,E1 -5862.945,E2 -5862.945} C_VEL
LIN {X 0,Y 504.194,Z 471.375,A -85,B 0,C 180,E1 -5863.502,E2 -5863.502} C_VEL
LIN {X 0,Y 504.352,Z 459.104,A -85,B 0,C 180,E1 -5863.896,E2 -5863.896} C_VEL
LIN {X 0,Y 502.91,Z 447.001,A -85,B 0,C 180,E1 -5864.181,E2 -5864.181} C_VEL
LIN {X 0,Y 503.329,Z 430.093,A -85,B 0,C 180,E1 -5867.26,E2 -5867.26} C_VEL
LIN {X 0,Y 503.74,Z 413.72,A -85,B 0,C 180,E1 -5870.2,E2 -5870.2} C_VEL
LIN {X 0,Y 504.337,Z 399.264,A -85,B 0,C 180,E1 -5872.966,E2 -5872.966} C_VEL
LIN {X 0,Y 505.085,Z 382.55,A -85,B 0,C 180,E1 -5876.218,E2 -5876.218} C_VEL
LIN {X 0,Y 505.646,Z 372.572,A -85,B 0,C 180,E1 -5878.201,E2 -5878.201} C_VEL
LIN {X 0,Y 504.619,Z 365.945,A -85,B 0,C 180,E1 -5879.631,E2 -5879.631} C_VEL
LIN {X 0,Y 502.796,Z 357.857,A -85,B 0,C 180,E1 -5881.499,E2 -5881.499} C_VEL
LIN {X 0,Y 502.806,Z 357.855,A -85,B 0,C 180,E1 -5883.994,E2 -5883.994} C_VEL
LIN {X 0,Y 502.779,Z 357.857,A -85,B 0,C 180,E1 -5887.178,E2 -5887.178} C_VEL
LIN {X 0,Y 502.789,Z 357.858,A -85,B 0,C 180,E1 -5890.015,E2 -5890.015} C_VEL
LIN {X 0,Y 502.804,Z 357.854,A -85,B 0,C 180,E1 -5892.199,E2 -5892.199} C_VEL
LIN {X 0,Y 502.802,Z 357.856,A -85,B 0,C 180,E1 -5895.468,E2 -5895.468} C_VEL
LIN {X 0,Y 502.831,Z 357.849,A -85,B 0,C 180,E1 -5897.864,E2 -5897.864} C_VEL
LIN {X 0,Y 502.804,Z 357.851,A -85,B 0,C 180,E1 -5901.024,E2 -5901.024} C_VEL
LIN {X 0,Y 502.785,Z 357.855,A -85,B 0,C 180,E1 -5904.167,E2 -5904.167} C_VEL
LIN {X 0,Y 502.834,Z 357.852,A -85,B 0,C 180,E1 -5906.993,E2 -5906.993} C_VEL
LIN {X 0,Y 502.816,Z 357.855,A -85,B 0,C 180,E1 -5910.065,E2 -5910.065} C_VEL
LIN {X 0,Y 502.836,Z 357.848,A -85,B 0,C 180,E1 -5912.533,E2 -5912.533} C_VEL
LIN {X 0,Y 502.828,Z 357.853,A -85,B 0,C 180,E1 -5915.299,E2 -5915.299} C_VEL
LIN {X 0,Y 502.781,Z 357.856,A -85,B 0,C 180,E1 -5917.826,E2 -5917.826} C_VEL
LIN {X 0,Y 502.826,Z 357.852,A -85,B 0,C 180,E1 -5920.4,E2 -5920.4} C_VEL
LIN {X 0,Y 502.836,Z 357.847,A -85,B 0,C 180,E1 -5922.932,E2 -5922.932} C_VEL
LIN {X 0,Y 502.854,Z 357.85,A -85,B 0,C 180,E1 -5925.429,E2 -5925.429} C_VEL
LIN {X 0,Y 502.879,Z 357.846,A -85,B 0,C 180,E1 -5928.717,E2 -5928.717} C_VEL
LIN {X 0,Y 502.903,Z 357.843,A -85,B 0,C 180,E1 -5931.967,E2 -5931.967} C_VEL
LIN {X 0,Y 502.939,Z 357.834,A -85,B 0,C 180,E1 -5934.387,E2 -5934.387} C_VEL
LIN {X 0,Y 503.026,Z 357.825,A -85,B 0,C 180,E1 -5937.598,E2 -5937.598} C_VEL
LIN {X 0,Y 503.029,Z 357.828,A -85,B 0,C 180,E1 -5940,E2 -5940} C_VEL
LIN {X 0,Y 503.027,Z 357.825,A -85,B 0,C 180,E1 -5942.402,E2 -5942.402} C_VEL
LIN {X 0,Y 502.94,Z 357.837,A -85,B 0,C 180,E1 -5945.614,E2 -5945.614} C_VEL
LIN {X 0,Y 502.904,Z 357.841,A -85,B 0,C 180,E1 -5948.033,E2 -5948.033} C_VEL
LIN {X 0,Y 502.894,Z 357.842,A -85,B 0,C 180,E1 -5951.283,E2 -5951.283} C_VEL
LIN {X 0,Y 502.847,Z 357.846,A -85,B 0,C 180,E1 -5954.571,E2 -5954.571} C_VEL
LIN {X 0,Y 502.864,Z 357.845,A -85,B 0,C 180,E1 -5957.907,E2 -5957.907} C_VEL
LIN {X 0,Y 502.83,Z 357.853,A -85,B 0,C 180,E1 -5960.536,E2 -5960.536} C_VEL
LIN {X 0,Y 502.799,Z 357.854,A -85,B 0,C 180,E1 -5963.04,E2 -5963.04} C_VEL
LIN {X 0,Y 502.842,Z 357.848,A -85,B 0,C 180,E1 -5965.676,E2 -5965.676} C_VEL
LIN {X 0,Y 502.841,Z 357.849,A -85,B 0,C 180,E1 -5968.373,E2 -5968.373} C_VEL
LIN {X 0,Y 502.795,Z 357.855,A -85,B 0,C 180,E1 -5971.499,E2 -5971.499} C_VEL
LIN {X 0,Y 502.806,Z 357.852,A -85,B 0,C 180,E1 -5974.444,E2 -5974.444} C_VEL
LIN {X 0,Y 502.782,Z 357.857,A -85,B 0,C 180,E1 -5977.178,E2 -5977.178} C_VEL
LIN {X 0,Y 502.79,Z 357.856,A -85,B 0,C 180,E1 -5980.015,E2 -5980.015} C_VEL
LIN {X 0,Y 502.804,Z 357.856,A -85,B 0,C 180,E1 -5982.199,E2 -5982.199} C_VEL
LIN {X 0,Y 502.803,Z 357.855,A -85,B 0,C 180,E1 -5985.468,E2 -5985.468} C_VEL
LIN {X 0,Y 502.832,Z 357.848,A -85,B 0,C 180,E1 -5987.864,E2 -5987.864} C_VEL
LIN {X 0,Y 502.803,Z 357.852,A -85,B 0,C 180,E1 -5991.024,E2 -5991.024} C_VEL
LIN {X 0,Y 502.777,Z 357.857,A -85,B 0,C 180,E1 -5994.169,E2 -5994.169} C_VEL
LIN {X 0,Y 502.811,Z 357.853,A -85,B 0,C 180,E1 -5997.223,E2 -5997.223} C_VEL
LIN {X 0,Y 502.109,Z 357.939,A -85,B 0,C 180,E1 -5997.891,E2 -5997.891} C_VEL
LIN {X 0,Y 499.245,Z 358.297,A -85,B 0,C 180,E1 -5998.977,E2 -5998.977} C_VEL
LIN {X 0,Y 496.85,Z 358.595,A -85,B 0,C 180,E1 -5999.852,E2 -5999.852} C_VEL
LIN {X 0,Y 495.834,Z 358.724,A -85,B 0,C 180,E1 -6000.528,E2 -6000.528} C_VEL
LIN {X 0,Y 495.756,Z 358.729,A -85,B 0,C 180,E1 -6000.756,E2 -6000.756} C_VEL
LIN {X 0,Y 495.794,Z 358.729,A -85,B 0,C 180,E1 -6003.932,E2 -6003.932} C_VEL
LIN {X 0,Y 495.763,Z 358.732,A -85,B 0,C 180,E1 -6007.139,E2 -6007.139} C_VEL
LIN {X 0,Y 495.782,Z 358.729,A -85,B 0,C 180,E1 -6010.11,E2 -6010.11} C_VEL
LIN {X 0,Y 495.79,Z 358.726,A -85,B 0,C 180,E1 -6012.682,E2 -6012.682} C_VEL
LIN {X 0,Y 495.793,Z 358.728,A -85,B 0,C 180,E1 -6015.217,E2 -6015.217} C_VEL
LIN {X 0,Y 495.855,Z 358.722,A -85,B 0,C 180,E1 -6018.555,E2 -6018.555} C_VEL
LIN {X 0,Y 495.876,Z 358.717,A -85,B 0,C 180,E1 -6021.852,E2 -6021.852} C_VEL
LIN {X 0,Y 495.894,Z 358.714,A -85,B 0,C 180,E1 -6024.307,E2 -6024.307} C_VEL
LIN {X 0,Y 495.997,Z 358.702,A -85,B 0,C 180,E1 -6027.564,E2 -6027.564} C_VEL
LIN {X 0,Y 496.003,Z 358.701,A -85,B 0,C 180,E1 -6030,E2 -6030} C_VEL
LIN {X 0,Y 495.997,Z 358.701,A -85,B 0,C 180,E1 -6032.436,E2 -6032.436} C_VEL
LIN {X 0,Y 495.893,Z 358.716,A -85,B 0,C 180,E1 -6035.694,E2 -6035.694} C_VEL
LIN {X 0,Y 495.877,Z 358.716,A -85,B 0,C 180,E1 -6038.148,E2 -6038.148} C_VEL
LIN {X 0,Y 495.856,Z 358.718,A -85,B 0,C 180,E1 -6041.445,E2 -6041.445} C_VEL
LIN {X 0,Y 495.794,Z 358.725,A -85,B 0,C 180,E1 -6044.783,E2 -6044.783} C_VEL
LIN {X 0,Y 495.786,Z 358.73,A -85,B 0,C 180,E1 -6047.319,E2 -6047.319} C_VEL
LIN {X 0,Y 495.775,Z 358.729,A -85,B 0,C 180,E1 -6049.89,E2 -6049.89} C_VEL
LIN {X 0,Y 495.763,Z 358.729,A -85,B 0,C 180,E1 -6052.861,E2 -6052.861} C_VEL
LIN {X 0,Y 495.784,Z 358.726,A -85,B 0,C 180,E1 -6056.068,E2 -6056.068} C_VEL
LIN {X 0,Y 495.776,Z 358.731,A -85,B 0,C 180,E1 -6058.815,E2 -6058.815} C_VEL
LIN {X 0,Y 495.76,Z 358.732,A -85,B 0,C 180,E1 -6061.726,E2 -6061.726} C_VEL
LIN {X 0,Y 495.772,Z 358.727,A -85,B 0,C 180,E1 -6064.694,E2 -6064.694} C_VEL
LIN {X 0,Y 495.732,Z 358.734,A -85,B 0,C 180,E1 -6067.562,E2 -6067.562} C_VEL
LIN {X 0,Y 495.77,Z 358.732,A -85,B 0,C 180,E1 -6070.7,E2 -6070.7} C_VEL
LIN {X 0,Y 495.735,Z 358.737,A -85,B 0,C 180,E1 -6073.695,E2 -6073.695} C_VEL
LIN {X 0,Y 495.729,Z 358.732,A -85,B 0,C 180,E1 -6076.306,E2 -6076.306} C_VEL
LIN {X 0,Y 495.77,Z 358.73,A -85,B 0,C 180,E1 -6079.3,E2 -6079.3} C_VEL
LIN {X 0,Y 495.735,Z 358.736,A -85,B 0,C 180,E1 -6082.439,E2 -6082.439} C_VEL
LIN {X 0,Y 495.787,Z 358.73,A -85,B 0,C 180,E1 -6085.457,E2 -6085.457} C_VEL
LIN {X 0,Y 495.76,Z 358.731,A -85,B 0,C 180,E1 -6088.364,E2 -6088.364} C_VEL
LIN {X 0,Y 495.867,Z 358.795,A -85,B 0,C 180,E1 -6089.833,E2 -6089.833} C_VEL
LIN {X 0,Y 495.703,Z 365.43,A -85,B 0,C 180,E1 -6093.019,E2 -6093.019} C_VEL
LIN {X 0,Y 495.582,Z 371.107,A -85,B 0,C 180,E1 -6095.716,E2 -6095.716} C_VEL
LIN {X 0,Y 495.465,Z 376.712,A -85,B 0,C 180,E1 -6098.358,E2 -6098.358} C_VEL
LIN {X 0,Y 495.409,Z 382.299,A -85,B 0,C 180,E1 -6100.957,E2 -6100.957} C_VEL
LIN {X 0,Y 495.315,Z 387.856,A -85,B 0,C 180,E1 -6103.514,E2 -6103.514} C_VEL
LIN {X 0,Y 495.207,Z 393.335,A -85,B 0,C 180,E1 -6106.039,E2 -6106.039} C_VEL
LIN {X 0,Y 495.198,Z 398.859,A -85,B 0,C 180,E1 -6108.539,E2 -6108.539} C_VEL
LIN {X 0,Y 495.147,Z 405.366,A -85,B 0,C 180,E1 -6111.429,E2 -6111.429} C_VEL
LIN {X 0,Y 496.134,Z 414.114,A -85,B 0,C 180,E1 -6111.805,E2 -6111.805} C_VEL
LIN {X 0,Y 496.009,Z 423.931,A -85,B 0,C 180,E1 -6112.367,E2 -6112.367} C_VEL
LIN {X 0,Y 495.83,Z 432.175,A -85,B 0,C 180,E1 -6113.003,E2 -6113.003} C_VEL
LIN {X 0,Y 495.569,Z 439.14,A -85,B 0,C 180,E1 -6113.69,E2 -6113.69} C_VEL
LIN {X 0,Y 495.539,Z 445.623,A -85,B 0,C 180,E1 -6114.507,E2 -6114.507} C_VEL
LIN {X 0,Y 495.448,Z 451.844,A -85,B 0,C 180,E1 -6115.525,E2 -6115.525} C_VEL
LIN {X 0,Y 495.406,Z 455.632,A -85,B 0,C 180,E1 -6116.34,E2 -6116.34} C_VEL
LIN {X 0,Y 495.294,Z 458.565,A -85,B 0,C 180,E1 -6117.153,E2 -6117.153} C_VEL
LIN {X 0,Y 495.059,Z 461.528,A -85,B 0,C 180,E1 -6118.373,E2 -6118.373} C_VEL
LIN {X 0,Y 495.039,Z 462.618,A -85,B 0,C 180,E1 -6119.187,E2 -6119.187} C_VEL
LIN {X 0,Y 495.039,Z 463.039,A -85,B 0,C 180,E1 -6120,E2 -6120} C_VEL
LIN {X 0,Y 495.048,Z 462.799,A -85,B 0,C 180,E1 -6120.813,E2 -6120.813} C_VEL
LIN {X 0,Y 495.077,Z 461.893,A -85,B 0,C 180,E1 -6121.627,E2 -6121.627} C_VEL
LIN {X 0,Y 495.298,Z 459.216,A -85,B 0,C 180,E1 -6122.847,E2 -6122.847} C_VEL
LIN {X 0,Y 495.445,Z 456.489,A -85,B 0,C 180,E1 -6123.66,E2 -6123.66} C_VEL
LIN {X 0,Y 495.478,Z 451.901,A -85,B 0,C 180,E1 -6124.678,E2 -6124.678} C_VEL
LIN {X 0,Y 495.614,Z 447.065,A -85,B 0,C 180,E1 -6125.493,E2 -6125.493} C_VEL
LIN {X 0,Y 495.721,Z 440.94,A -85,B 0,C 180,E1 -6126.308,E2 -6126.308} C_VEL
LIN {X 0,Y 495.917,Z 434.657,A -85,B 0,C 180,E1 -6126.975,E2 -6126.975} C_VEL
LIN {X 0,Y 496.104,Z 425.999,A -85,B 0,C 180,E1 -6127.693,E2 -6127.693} C_VEL
LIN {X 0,Y 496.318,Z 416.165,A -85,B 0,C 180,E1 -6128.294,E2 -6128.294} C_VEL
LIN {X 0,Y 495.792,Z 409.543,A -85,B 0,C 180,E1 -6128.611,E2 -6128.611} C_VEL
LIN {X 0,Y 495.294,Z 406.521,A -85,B 0,C 180,E1 -6128.748,E2 -6128.748} C_VEL
LIN {X 0,Y 495.359,Z 398.842,A -85,B 0,C 180,E1 -6132.287,E2 -6132.287} C_VEL
LIN {X 0,Y 495.509,Z 391.736,A -85,B 0,C 180,E1 -6135.634,E2 -6135.634} C_VEL
LIN {X 0,Y 495.626,Z 384.59,A -85,B 0,C 180,E1 -6139.035,E2 -6139.035} C_VEL
LIN {X 0,Y 495.765,Z 379.22,A -85,B 0,C 180,E1 -6141.628,E2 -6141.628} C_VEL
LIN {X 0,Y 495.926,Z 373.829,A -85,B 0,C 180,E1 -6144.266,E2 -6144.266} C_VEL
LIN {X 0,Y 496.072,Z 368.315,A -85,B 0,C 180,E1 -6146.959,E2 -6146.959} C_VEL
LIN {X 0,Y 496.252,Z 362.912,A -85,B 0,C 180,E1 -6149.714,E2 -6149.714} C_VEL
LIN {X 0,Y 495.788,Z 358.803,A -85,B 0,C 180,E1 -6151.886,E2 -6151.886} C_VEL
LIN {X 0,Y 495.772,Z 358.733,A -85,B 0,C 180,E1 -6154.694,E2 -6154.694} C_VEL
LIN {X 0,Y 495.734,Z 358.737,A -85,B 0,C 180,E1 -6157.561,E2 -6157.561} C_VEL
LIN {X 0,Y 495.797,Z 358.73,A -85,B 0,C 180,E1 -6160.052,E2 -6160.052} C_VEL
LIN {X 0,Y 495.767,Z 358.733,A -85,B 0,C 180,E1 -6162.879,E2 -6162.879} C_VEL
LIN {X 0,Y 495.74,Z 358.735,A -85,B 0,C 180,E1 -6165.999,E2 -6165.999} C_VEL
LIN {X 0,Y 495.766,Z 358.734,A -85,B 0,C 180,E1 -6168.706,E2 -6168.706} C_VEL
LIN {X 0,Y 495.753,Z 358.736,A -85,B 0,C 180,E1 -6171.408,E2 -6171.408} C_VEL
LIN {X 0,Y 495.751,Z 358.735,A -85,B 0,C 180,E1 -6174.462,E2 -6174.462} C_VEL
LIN {X 0,Y 495.846,Z 358.935,A -85,B 0,C 180,E1 -6177.086,E2 -6177.086} C_VEL
LIN {X 0,Y 497.613,Z 366.809,A -85,B 0,C 180,E1 -6179.489,E2 -6179.489} C_VEL
LIN {X 0,Y 499.031,Z 373.916,A -85,B 0,C 180,E1 -6181.391,E2 -6181.391} C_VEL
LIN {X 0,Y 498.435,Z 381.779,A -85,B 0,C 180,E1 -6183.179,E2 -6183.179} C_VEL
LIN {X 0,Y 497.466,Z 396.359,A -85,B 0,C 180,E1 -6186.257,E2 -6186.257} C_VEL
LIN {X 0,Y 496.708,Z 412.818,A -85,B 0,C 180,E1 -6189.501,E2 -6189.501} C_VEL
LIN {X 0,Y 496.197,Z 428.687,A -85,B 0,C 180,E1 -6192.483,E2 -6192.483} C_VEL
LIN {X 0,Y 495.821,Z 445.977,A -85,B 0,C 180,E1 -6195.637,E2 -6195.637} C_VEL
LIN {X 0,Y 495.805,Z 446.267,A -85,B 0,C 180,E1 -6195.689,E2 -6195.689} C_VEL
LIN {X 0,Y 497.211,Z 458.713,A -85,B 0,C 180,E1 -6195.979,E2 -6195.979} C_VEL
LIN {X 0,Y 497.168,Z 471.597,A -85,B 0,C 180,E1 -6196.407,E2 -6196.407} C_VEL
LIN {X 0,Y 496.846,Z 483.898,A -85,B 0,C 180,E1 -6196.976,E2 -6196.976} C_VEL
LIN {X 0,Y 496.511,Z 496.249,A -85,B 0,C 180,E1 -6197.741,E2 -6197.741} C_VEL
LIN {X 0,Y 496.125,Z 507.925,A -85,B 0,C 180,E1 -6198.665,E2 -6198.665} C_VEL
LIN {X 0,Y 495.852,Z 517.296,A -85,B 0,C 180,E1 -6199.589,E2 -6199.589} C_VEL
LIN {X 0,Y 495.601,Z 525.832,A -85,B 0,C 180,E1 -6200.614,E2 -6200.614} C_VEL
LIN {X 0,Y 495.397,Z 534.173,A -85,B 0,C 180,E1 -6201.844,E2 -6201.844} C_VEL
LIN {X 0,Y 495.251,Z 540.878,A -85,B 0,C 180,E1 -6203.072,E2 -6203.072} C_VEL
LIN {X 0,Y 495.218,Z 546.199,A -85,B 0,C 180,E1 -6204.299,E2 -6204.299} C_VEL
LIN {X 0,Y 495.095,Z 550.306,A -85,B 0,C 180,E1 -6205.522,E2 -6205.522} C_VEL
LIN {X 0,Y 495.116,Z 553.348,A -85,B 0,C 180,E1 -6206.745,E2 -6206.745} C_VEL
LIN {X 0,Y 495.058,Z 554.796,A -85,B 0,C 180,E1 -6207.559,E2 -6207.559} C_VEL
LIN {X 0,Y 494.951,Z 556.457,A -85,B 0,C 180,E1 -6209.186,E2 -6209.186} C_VEL
LIN {X 0,Y 494.948,Z 556.692,A -85,B 0,C 180,E1 -6210,E2 -6210} C_VEL
LIN {X 0,Y 494.95,Z 556.478,A -85,B 0,C 180,E1 -6210.813,E2 -6210.813} C_VEL
LIN {X 0,Y 495.058,Z 554.865,A -85,B 0,C 180,E1 -6212.441,E2 -6212.441} C_VEL
LIN {X 0,Y 495.116,Z 553.437,A -85,B 0,C 180,E1 -6213.255,E2 -6213.255} C_VEL
LIN {X 0,Y 495.076,Z 550.43,A -85,B 0,C 180,E1 -6214.478,E2 -6214.478} C_VEL
LIN {X 0,Y 495.188,Z 545.213,A -85,B 0,C 180,E1 -6215.988,E2 -6215.988} C_VEL
LIN {X 0,Y 495.274,Z 539.044,A -85,B 0,C 180,E1 -6217.337,E2 -6217.337} C_VEL
LIN {X 0,Y 495.454,Z 531.915,A -85,B 0,C 180,E1 -6218.565,E2 -6218.565} C_VEL
LIN {X 0,Y 495.659,Z 522.976,A -85,B 0,C 180,E1 -6219.796,E2 -6219.796} C_VEL
LIN {X 0,Y 495.977,Z 513.814,A -85,B 0,C 180,E1 -6220.822,E2 -6220.822} C_VEL
LIN {X 0,Y 496.317,Z 503.661,A -85,B 0,C 180,E1 -6221.745,E2 -6221.745} C_VEL
LIN {X 0,Y 496.661,Z 492.511,A -85,B 0,C 180,E1 -6222.555,E2 -6222.555} C_VEL
LIN {X 0,Y 496.975,Z 480.639,A -85,B 0,C 180,E1 -6223.233,E2 -6223.233} C_VEL
LIN {X 0,Y 497.29,Z 467.921,A -85,B 0,C 180,E1 -6223.771,E2 -6223.771} C_VEL
LIN {X 0,Y 497.219,Z 458.253,A -85,B 0,C 180,E1 -6224.073,E2 -6224.073} C_VEL
LIN {X 0,Y 495.893,Z 446.63,A -85,B 0,C 180,E1 -6224.36,E2 -6224.36} C_VEL
LIN {X 0,Y 496.334,Z 428.595,A -85,B 0,C 180,E1 -6227.724,E2 -6227.724} C_VEL
LIN {X 0,Y 496.743,Z 414.657,A -85,B 0,C 180,E1 -6230.281,E2 -6230.281} C_VEL
LIN {X 0,Y 497.392,Z 399.67,A -85,B 0,C 180,E1 -6233.19,E2 -6233.19} C_VEL
LIN {X 0,Y 498.211,Z 383.54,A -85,B 0,C 180,E1 -6236.382,E2 -6236.382} C_VEL
LIN {X 0,Y 498.76,Z 373.61,A -85,B 0,C 180,E1 -6238.396,E2 -6238.396} C_VEL
LIN {X 0,Y 497.414,Z 366.338,A -85,B 0,C 180,E1 -6240.01,E2 -6240.01} C_VEL
LIN {X 0,Y 495.745,Z 358.736,A -85,B 0,C 180,E1 -6241.767,E2 -6241.767} C_VEL
LIN {X 0,Y 495.771,Z 358.731,A -85,B 0,C 180,E1 -6244.694,E2 -6244.694} C_VEL
LIN {X 0,Y 495.73,Z 358.733,A -85,B 0,C 180,E1 -6247.561,E2 -6247.561} C_VEL
LIN {X 0,Y 495.768,Z 358.729,A -85,B 0,C 180,E1 -6250.7,E2 -6250.7} C_VEL
LIN {X 0,Y 495.737,Z 358.737,A -85,B 0,C 180,E1 -6253.695,E2 -6253.695} C_VEL
LIN {X 0,Y 495.736,Z 358.734,A -85,B 0,C 180,E1 -6256.304,E2 -6256.304} C_VEL
LIN {X 0,Y 495.768,Z 358.728,A -85,B 0,C 180,E1 -6259.3,E2 -6259.3} C_VEL
LIN {X 0,Y 495.733,Z 358.733,A -85,B 0,C 180,E1 -6262.439,E2 -6262.439} C_VEL
LIN {X 0,Y 495.785,Z 358.73,A -85,B 0,C 180,E1 -6265.457,E2 -6265.457} C_VEL
LIN {X 0,Y 495.757,Z 358.735,A -85,B 0,C 180,E1 -6268.364,E2 -6268.364} C_VEL
LIN {X 0,Y 495.789,Z 358.727,A -85,B 0,C 180,E1 -6271.507,E2 -6271.507} C_VEL
LIN {X 0,Y 495.792,Z 358.728,A -85,B 0,C 180,E1 -6273.932,E2 -6273.932} C_VEL
LIN {X 0,Y 495.761,Z 358.733,A -85,B 0,C 180,E1 -6277.139,E2 -6277.139} C_VEL
LIN {X 0,Y 495.78,Z 358.732,A -85,B 0,C 180,E1 -6280.11,E2 -6280.11} C_VEL
LIN {X 0,Y 495.788,Z 358.725,A -85,B 0,C 180,E1 -6282.681,E2 -6282.681} C_VEL
LIN {X 0,Y 495.796,Z 358.729,A -85,B 0,C 180,E1 -6285.217,E2 -6285.217} C_VEL
LIN {X 0,Y 495.854,Z 358.721,A -85,B 0,C 180,E1 -6288.555,E2 -6288.555} C_VEL
LIN {X 0,Y 495.875,Z 358.72,A -85,B 0,C 180,E1 -6291.852,E2 -6291.852} C_VEL
LIN {X 0,Y 495.897,Z 358.712,A -85,B 0,C 180,E1 -6294.307,E2 -6294.307} C_VEL
LIN {X 0,Y 495.995,Z 358.701,A -85,B 0,C 180,E1 -6297.564,E2 -6297.564} C_VEL
LIN {X 0,Y 496.001,Z 358.703,A -85,B 0,C 180,E1 -6300,E2 -6300} C_VEL
LIN {X 0,Y 495.995,Z 358.701,A -85,B 0,C 180,E1 -6302.436,E2 -6302.436} C_VEL
LIN {X 0,Y 495.898,Z 358.713,A -85,B 0,C 180,E1 -6305.693,E2 -6305.693} C_VEL
LIN {X 0,Y 495.875,Z 358.717,A -85,B 0,C 180,E1 -6308.148,E2 -6308.148} C_VEL
LIN {X 0,Y 495.869,Z 358.718,A -85,B 0,C 180,E1 -6311.445,E2 -6311.445} C_VEL
LIN {X 0,Y 495.792,Z 358.726,A -85,B 0,C 180,E1 -6314.783,E2 -6314.783} C_VEL
LIN {X 0,Y 495.788,Z 358.728,A -85,B 0,C 180,E1 -6317.319,E2 -6317.319} C_VEL
LIN {X 0,Y 495.78,Z 358.729,A -85,B 0,C 180,E1 -6319.89,E2 -6319.89} C_VEL
LIN {X 0,Y 495.767,Z 358.729,A -85,B 0,C 180,E1 -6322.863,E2 -6322.863} C_VEL
LIN {X 0,Y 495.792,Z 358.724,A -85,B 0,C 180,E1 -6326.068,E2 -6326.068} C_VEL
LIN {X 0,Y 495.773,Z 358.732,A -85,B 0,C 180,E1 -6328.815,E2 -6328.815} C_VEL
LIN {X 0,Y 495.758,Z 358.733,A -85,B 0,C 180,E1 -6331.726,E2 -6331.726} C_VEL
LIN {X 0,Y 495.776,Z 358.728,A -85,B 0,C 180,E1 -6334.695,E2 -6334.695} C_VEL
LIN {X 0,Y 495.732,Z 358.732,A -85,B 0,C 180,E1 -6337.562,E2 -6337.562} C_VEL
LIN {X 0,Y 495.769,Z 358.731,A -85,B 0,C 180,E1 -6340.7,E2 -6340.7} C_VEL
LIN {X 0,Y 495.735,Z 358.735,A -85,B 0,C 180,E1 -6344.001,E2 -6344.001} C_VEL
LIN {X 0,Y 495.735,Z 358.735,A -85,B 0,C 180,E1 -6347.118,E2 -6347.118} C_VEL
LIN {X 0,Y 495.76,Z 358.73,A -85,B 0,C 180,E1 -6349.953,E2 -6349.953} C_VEL
LIN {X 0,Y 495.73,Z 358.735,A -85,B 0,C 180,E1 -6352.553,E2 -6352.553} C_VEL
LIN {X 0,Y 495.78,Z 358.73,A -85,B 0,C 180,E1 -6355.457,E2 -6355.457} C_VEL
LIN {X 0,Y 495.759,Z 358.732,A -85,B 0,C 180,E1 -6358.364,E2 -6358.364} C_VEL
LIN {X 0,Y 495.756,Z 358.729,A -85,B 0,C 180,E1 -6360.756,E2 -6360.756} C_VEL
LIN {X 0,Y 495.098,Z 358.813,A -85,B 0,C 180,E1 -6361.435,E2 -6361.435} C_VEL
LIN {X 0,Y 492.242,Z 359.169,A -85,B 0,C 180,E1 -6362.538,E2 -6362.538} C_VEL
LIN {X 0,Y 489.833,Z 359.47,A -85,B 0,C 180,E1 -6363.427,E2 -6363.427} C_VEL
LIN {X 0,Y 488.817,Z 359.597,A -85,B 0,C 180,E1 -6364.113,E2 -6364.113} C_VEL
LIN {X 0,Y 488.745,Z 359.604,A -85,B 0,C 180,E1 -6364.345,E2 -6364.345} C_VEL
LIN {X 0,Y 488.725,Z 359.608,A -85,B 0,C 180,E1 -6367.153,E2 -6367.153} C_VEL
LIN {X 0,Y 488.732,Z 359.605,A -85,B 0,C 180,E1 -6369.811,E2 -6369.811} C_VEL
LIN {X 0,Y 488.737,Z 359.606,A -85,B 0,C 180,E1 -6372.424,E2 -6372.424} C_VEL
LIN {X 0,Y 488.765,Z 359.603,A -85,B 0,C 180,E1 -6375,E2 -6375} C_VEL
LIN {X 0,Y 488.809,Z 359.598,A -85,B 0,C 180,E1 -6378.388,E2 -6378.388} C_VEL
LIN {X 0,Y 488.82,Z 359.595,A -85,B 0,C 180,E1 -6381.734,E2 -6381.734} C_VEL
LIN {X 0,Y 488.852,Z 359.591,A -85,B 0,C 180,E1 -6384.224,E2 -6384.224} C_VEL
LIN {X 0,Y 488.964,Z 359.578,A -85,B 0,C 180,E1 -6387.529,E2 -6387.529} C_VEL
LIN {X 0,Y 488.958,Z 359.578,A -85,B 0,C 180,E1 -6390.824,E2 -6390.824} C_VEL
LIN {X 0,Y 488.964,Z 359.576,A -85,B 0,C 180,E1 -6392.472,E2 -6392.472} C_VEL
LIN {X 0,Y 488.851,Z 359.593,A -85,B 0,C 180,E1 -6395.776,E2 -6395.776} C_VEL
LIN {X 0,Y 488.821,Z 359.596,A -85,B 0,C 180,E1 -6398.266,E2 -6398.266} C_VEL
LIN {X 0,Y 488.81,Z 359.597,A -85,B 0,C 180,E1 -6401.613,E2 -6401.613} C_VEL
LIN {X 0,Y 488.766,Z 359.601,A -85,B 0,C 180,E1 -6405,E2 -6405} C_VEL
LIN {X 0,Y 488.759,Z 359.605,A -85,B 0,C 180,E1 -6408.442,E2 -6408.442} C_VEL
LIN {X 0,Y 488.71,Z 359.609,A -85,B 0,C 180,E1 -6411.071,E2 -6411.071} C_VEL
LIN {X 0,Y 488.684,Z 359.616,A -85,B 0,C 180,E1 -6413.746,E2 -6413.746} C_VEL
LIN {X 0,Y 488.796,Z 359.599,A -85,B 0,C 180,E1 -6416.944,E2 -6416.944} C_VEL
LIN {X 0,Y 488.713,Z 359.61,A -85,B 0,C 180,E1 -6420.363,E2 -6420.363} C_VEL
LIN {X 0,Y 488.738,Z 359.607,A -85,B 0,C 180,E1 -6423.484,E2 -6423.484} C_VEL
LIN {X 0,Y 488.685,Z 359.61,A -85,B 0,C 180,E1 -6426.355,E2 -6426.355} C_VEL
LIN {X 0,Y 488.704,Z 359.61,A -85,B 0,C 180,E1 -6429.254,E2 -6429.254} C_VEL
LIN {X 0,Y 488.727,Z 359.607,A -85,B 0,C 180,E1 -6431.602,E2 -6431.602} C_VEL
LIN {X 0,Y 488.705,Z 359.609,A -85,B 0,C 180,E1 -6434.803,E2 -6434.803} C_VEL
LIN {X 0,Y 488.695,Z 359.611,A -85,B 0,C 180,E1 -6437.475,E2 -6437.475} C_VEL
LIN {X 0,Y 488.736,Z 359.605,A -85,B 0,C 180,E1 -6439.677,E2 -6439.677} C_VEL
LIN {X 0,Y 488.686,Z 359.612,A -85,B 0,C 180,E1 -6442.841,E2 -6442.841} C_VEL
LIN {X 0,Y 488.737,Z 359.605,A -85,B 0,C 180,E1 -6445.888,E2 -6445.888} C_VEL
LIN {X 0,Y 488.733,Z 359.612,A -85,B 0,C 180,E1 -6448.823,E2 -6448.823} C_VEL
LIN {X 0,Y 488.822,Z 359.682,A -85,B 0,C 180,E1 -6449.787,E2 -6449.787} C_VEL
LIN {X 0,Y 488.67,Z 366.484,A -85,B 0,C 180,E1 -6453.085,E2 -6453.085} C_VEL
LIN {X 0,Y 488.526,Z 373.092,A -85,B 0,C 180,E1 -6456.246,E2 -6456.246} C_VEL
LIN {X 0,Y 488.42,Z 379.515,A -85,B 0,C 180,E1 -6459.278,E2 -6459.278} C_VEL
LIN {X 0,Y 488.289,Z 386.192,A -85,B 0,C 180,E1 -6462.407,E2 -6462.407} C_VEL
LIN {X 0,Y 488.262,Z 391.794,A -85,B 0,C 180,E1 -6464.984,E2 -6464.984} C_VEL
LIN {X 0,Y 488.162,Z 399.214,A -85,B 0,C 180,E1 -6468.372,E2 -6468.372} C_VEL
LIN {X 0,Y 488.061,Z 405.663,A -85,B 0,C 180,E1 -6471.277,E2 -6471.277} C_VEL
LIN {X 0,Y 489.129,Z 413.838,A -85,B 0,C 180,E1 -6471.635,E2 -6471.635} C_VEL
LIN {X 0,Y 489.033,Z 423.059,A -85,B 0,C 180,E1 -6472.153,E2 -6472.153} C_VEL
LIN {X 0,Y 488.865,Z 431.875,A -85,B 0,C 180,E1 -6472.821,E2 -6472.821} C_VEL
LIN {X 0,Y 488.543,Z 439.748,A -85,B 0,C 180,E1 -6473.599,E2 -6473.599} C_VEL
LIN {X 0,Y 488.518,Z 446.237,A -85,B 0,C 180,E1 -6474.427,E2 -6474.427} C_VEL
LIN {X 0,Y 488.418,Z 452.458,A -85,B 0,C 180,E1 -6475.461,E2 -6475.461} C_VEL
LIN {X 0,Y 488.347,Z 456.257,A -85,B 0,C 180,E1 -6476.287,E2 -6476.287} C_VEL
LIN {X 0,Y 488.253,Z 459.199,A -85,B 0,C 180,E1 -6477.112,E2 -6477.112} C_VEL
LIN {X 0,Y 487.994,Z 462.187,A -85,B 0,C 180,E1 -6478.349,E2 -6478.349} C_VEL
LIN {X 0,Y 487.973,Z 463.287,A -85,B 0,C 180,E1 -6479.175,E2 -6479.175} C_VEL
LIN {X 0,Y 487.973,Z 463.718,A -85,B 0,C 180,E1 -6480,E2 -6480} C_VEL
LIN {X 0,Y 487.983,Z 463.486,A -85,B 0,C 180,E1 -6480.825,E2 -6480.825} C_VEL
LIN {X 0,Y 488.015,Z 462.588,A -85,B 0,C 180,E1 -6481.65,E2 -6481.65} C_VEL
LIN {X 0,Y 488.258,Z 459.924,A -85,B 0,C 180,E1 -6482.888,E2 -6482.888} C_VEL
LIN {X 0,Y 488.414,Z 457.208,A -85,B 0,C 180,E1 -6483.713,E2 -6483.713} C_VEL
LIN {X 0,Y 488.454,Z 452.643,A -85,B 0,C 180,E1 -6484.746,E2 -6484.746} C_VEL
LIN {X 0,Y 488.605,Z 447.83,A -85,B 0,C 180,E1 -6485.572,E2 -6485.572} C_VEL
LIN {X 0,Y 488.735,Z 441.754,A -85,B 0,C 180,E1 -6486.399,E2 -6486.399} C_VEL
LIN {X 0,Y 489.017,Z 433.891,A -85,B 0,C 180,E1 -6487.228,E2 -6487.228} C_VEL
LIN {X 0,Y 489.204,Z 424.935,A -85,B 0,C 180,E1 -6487.948,E2 -6487.948} C_VEL
LIN {X 0,Y 489.413,Z 415.35,A -85,B 0,C 180,E1 -6488.516,E2 -6488.516} C_VEL
LIN {X 0,Y 488.216,Z 406.94,A -85,B 0,C 180,E1 -6488.928,E2 -6488.928} C_VEL
LIN {X 0,Y 488.328,Z 399.373,A -85,B 0,C 180,E1 -6492.467,E2 -6492.467} C_VEL
LIN {X 0,Y 488.471,Z 392.205,A -85,B 0,C 180,E1 -6495.865,E2 -6495.865} C_VEL
LIN {X 0,Y 488.592,Z 386.853,A -85,B 0,C 180,E1 -6498.449,E2 -6498.449} C_VEL
LIN {X 0,Y 488.763,Z 379.694,A -85,B 0,C 180,E1 -6501.954,E2 -6501.954} C_VEL
LIN {X 0,Y 488.971,Z 373.317,A -85,B 0,C 180,E1 -6505.108,E2 -6505.108} C_VEL
LIN {X 0,Y 489.205,Z 367.053,A -85,B 0,C 180,E1 -6508.3,E2 -6508.3} C_VEL
LIN {X 0,Y 489.257,Z 362.94,A -85,B 0,C 180,E1 -6510.471,E2 -6510.471} C_VEL
LIN {X 0,Y 488.736,Z 359.61,A -85,B 0,C 180,E1 -6512.388,E2 -6512.388} C_VEL
LIN {X 0,Y 488.72,Z 359.611,A -85,B 0,C 180,E1 -6515.115,E2 -6515.115} C_VEL
LIN {X 0,Y 488.692,Z 359.615,A -85,B 0,C 180,E1 -6518.199,E2 -6518.199} C_VEL
LIN {X 0,Y 488.753,Z 359.606,A -85,B 0,C 180,E1 -6520.349,E2 -6520.349} C_VEL
LIN {X 0,Y 488.72,Z 359.61,A -85,B 0,C 180,E1 -6523.651,E2 -6523.651} C_VEL
LIN {X 0,Y 488.696,Z 359.615,A -85,B 0,C 180,E1 -6526.346,E2 -6526.346} C_VEL
LIN {X 0,Y 488.722,Z 359.611,A -85,B 0,C 180,E1 -6528.586,E2 -6528.586} C_VEL
LIN {X 0,Y 488.682,Z 359.616,A -85,B 0,C 180,E1 -6531.8,E2 -6531.8} C_VEL
LIN {X 0,Y 488.726,Z 359.612,A -85,B 0,C 180,E1 -6535.052,E2 -6535.052} C_VEL
LIN {X 0,Y 488.757,Z 359.788,A -85,B 0,C 180,E1 -6536.512,E2 -6536.512} C_VEL
LIN {X 0,Y 490.106,Z 365.606,A -85,B 0,C 180,E1 -6538.439,E2 -6538.439} C_VEL
LIN {X 0,Y 491.819,Z 373.246,A -85,B 0,C 180,E1 -6540.655,E2 -6540.655} C_VEL
LIN {X 0,Y 492.185,Z 376.18,A -85,B 0,C 180,E1 -6541.422,E2 -6541.422} C_VEL
LIN {X 0,Y 491.489,Z 384.027,A -85,B 0,C 180,E1 -6543.228,E2 -6543.228} C_VEL
LIN {X 0,Y 490.48,Z 398.419,A -85,B 0,C 180,E1 -6546.346,E2 -6546.346} C_VEL
LIN {X 0,Y 489.697,Z 414.784,A -85,B 0,C 180,E1 -6549.633,E2 -6549.633} C_VEL
LIN {X 0,Y 489.092,Z 431.646,A -85,B 0,C 180,E1 -6552.868,E2 -6552.868} C_VEL
LIN {X 0,Y 488.771,Z 445.854,A -85,B 0,C 180,E1 -6555.506,E2 -6555.506} C_VEL
LIN {X 0,Y 490.366,Z 461.794,A -85,B 0,C 180,E1 -6555.924,E2 -6555.924} C_VEL
LIN {X 0,Y 490.1,Z 473.88,A -85,B 0,C 180,E1 -6556.366,E2 -6556.366} C_VEL
LIN {X 0,Y 489.771,Z 485.658,A -85,B 0,C 180,E1 -6556.959,E2 -6556.959} C_VEL
LIN {X 0,Y 489.45,Z 498.13,A -85,B 0,C 180,E1 -6557.778,E2 -6557.778} C_VEL
LIN {X 0,Y 488.985,Z 509.165,A -85,B 0,C 180,E1 -6558.707,E2 -6558.707} C_VEL
LIN {X 0,Y 488.738,Z 518.212,A -85,B 0,C 180,E1 -6559.645,E2 -6559.645} C_VEL
LIN {X 0,Y 488.482,Z 526.505,A -85,B 0,C 180,E1 -6560.685,E2 -6560.685} C_VEL
LIN {X 0,Y 488.285,Z 534.627,A -85,B 0,C 180,E1 -6561.933,E2 -6561.933} C_VEL
LIN {X 0,Y 488.18,Z 540.111,A -85,B 0,C 180,E1 -6562.971,E2 -6562.971} C_VEL
LIN {X 0,Y 488.131,Z 545.468,A -85,B 0,C 180,E1 -6564.215,E2 -6564.215} C_VEL
LIN {X 0,Y 487.998,Z 549.599,A -85,B 0,C 180,E1 -6565.457,E2 -6565.457} C_VEL
LIN {X 0,Y 488.039,Z 552.66,A -85,B 0,C 180,E1 -6566.698,E2 -6566.698} C_VEL
LIN {X 0,Y 487.995,Z 554.12,A -85,B 0,C 180,E1 -6567.524,E2 -6567.524} C_VEL
LIN {X 0,Y 487.882,Z 555.795,A -85,B 0,C 180,E1 -6569.174,E2 -6569.174} C_VEL
LIN {X 0,Y 487.88,Z 556.033,A -85,B 0,C 180,E1 -6570,E2 -6570} C_VEL
LIN {X 0,Y 487.88,Z 555.82,A -85,B 0,C 180,E1 -6570.825,E2 -6570.825} C_VEL
LIN {X 0,Y 487.995,Z 554.21,A -85,B 0,C 180,E1 -6572.476,E2 -6572.476} C_VEL
LIN {X 0,Y 488.039,Z 552.774,A -85,B 0,C 180,E1 -6573.302,E2 -6573.302} C_VEL
LIN {X 0,Y 487.981,Z 549.758,A -85,B 0,C 180,E1 -6574.543,E2 -6574.543} C_VEL
LIN {X 0,Y 488.107,Z 545.676,A -85,B 0,C 180,E1 -6575.784,E2 -6575.784} C_VEL
LIN {X 0,Y 488.181,Z 539.36,A -85,B 0,C 180,E1 -6577.236,E2 -6577.236} C_VEL
LIN {X 0,Y 488.355,Z 532.471,A -85,B 0,C 180,E1 -6578.482,E2 -6578.482} C_VEL
LIN {X 0,Y 488.547,Z 525.423,A -85,B 0,C 180,E1 -6579.522,E2 -6579.522} C_VEL
LIN {X 0,Y 488.822,Z 516.919,A -85,B 0,C 180,E1 -6580.563,E2 -6580.563} C_VEL
LIN {X 0,Y 489.215,Z 506.381,A -85,B 0,C 180,E1 -6581.602,E2 -6581.602} C_VEL
LIN {X 0,Y 489.548,Z 494.768,A -85,B 0,C 180,E1 -6582.521,E2 -6582.521} C_VEL
LIN {X 0,Y 489.908,Z 482.476,A -85,B 0,C 180,E1 -6583.269,E2 -6583.269} C_VEL
LIN {X 0,Y 490.262,Z 469.982,A -85,B 0,C 180,E1 -6583.84,E2 -6583.84} C_VEL
LIN {X 0,Y 490.281,Z 459.298,A -85,B 0,C 180,E1 -6584.197,E2 -6584.197} C_VEL
LIN {X 0,Y 488.92,Z 447.494,A -85,B 0,C 180,E1 -6584.49,E2 -6584.49} C_VEL
LIN {X 0,Y 488.838,Z 446.397,A -85,B 0,C 180,E1 -6584.519,E2 -6584.519} C_VEL
LIN {X 0,Y 489.344,Z 428.137,A -85,B 0,C 180,E1 -6587.986,E2 -6587.986} C_VEL
LIN {X 0,Y 489.867,Z 413.373,A -85,B 0,C 180,E1 -6590.798,E2 -6590.798} C_VEL
LIN {X 0,Y 490.715,Z 395.583,A -85,B 0,C 180,E1 -6594.315,E2 -6594.315} C_VEL
LIN {X 0,Y 491.637,Z 379.46,A -85,B 0,C 180,E1 -6597.588,E2 -6597.588} C_VEL
LIN {X 0,Y 491.819,Z 374.592,A -85,B 0,C 180,E1 -6598.601,E2 -6598.601} C_VEL
LIN {X 0,Y 490.196,Z 366.28,A -85,B 0,C 180,E1 -6600.491,E2 -6600.491} C_VEL
LIN {X 0,Y 488.705,Z 359.612,A -85,B 0,C 180,E1 -6602.08,E2 -6602.08} C_VEL
LIN {X 0,Y 488.719,Z 359.612,A -85,B 0,C 180,E1 -6605.115,E2 -6605.115} C_VEL
LIN {X 0,Y 488.681,Z 359.613,A -85,B 0,C 180,E1 -6608.2,E2 -6608.2} C_VEL
LIN {X 0,Y 488.72,Z 359.608,A -85,B 0,C 180,E1 -6611.414,E2 -6611.414} C_VEL
LIN {X 0,Y 488.704,Z 359.61,A -85,B 0,C 180,E1 -6614.024,E2 -6614.024} C_VEL
LIN {X 0,Y 488.717,Z 359.609,A -85,B 0,C 180,E1 -6617.173,E2 -6617.173} C_VEL
LIN {X 0,Y 488.734,Z 359.605,A -85,B 0,C 180,E1 -6619.676,E2 -6619.676} C_VEL
LIN {X 0,Y 488.684,Z 359.611,A -85,B 0,C 180,E1 -6622.841,E2 -6622.841} C_VEL
LIN {X 0,Y 488.735,Z 359.606,A -85,B 0,C 180,E1 -6625.887,E2 -6625.887} C_VEL
LIN {X 0,Y 488.693,Z 359.611,A -85,B 0,C 180,E1 -6628.82,E2 -6628.82} C_VEL
LIN {X 0,Y 488.746,Z 359.605,A -85,B 0,C 180,E1 -6631.671,E2 -6631.671} C_VEL
LIN {X 0,Y 488.749,Z 359.603,A -85,B 0,C 180,E1 -6634.444,E2 -6634.444} C_VEL
LIN {X 0,Y 488.724,Z 359.61,A -85,B 0,C 180,E1 -6637.153,E2 -6637.153} C_VEL
LIN {X 0,Y 488.73,Z 359.607,A -85,B 0,C 180,E1 -6639.811,E2 -6639.811} C_VEL
LIN {X 0,Y 488.735,Z 359.604,A -85,B 0,C 180,E1 -6642.423,E2 -6642.423} C_VEL
LIN {X 0,Y 488.767,Z 359.603,A -85,B 0,C 180,E1 -6645,E2 -6645} C_VEL
LIN {X 0,Y 488.807,Z 359.599,A -85,B 0,C 180,E1 -6648.388,E2 -6648.388} C_VEL
LIN {X 0,Y 488.819,Z 359.598,A -85,B 0,C 180,E1 -6651.734,E2 -6651.734} C_VEL
LIN {X 0,Y 488.856,Z 359.589,A -85,B 0,C 180,E1 -6654.224,E2 -6654.224} C_VEL
LIN {X 0,Y 488.963,Z 359.577,A -85,B 0,C 180,E1 -6657.529,E2 -6657.529} C_VEL
LIN {X 0,Y 488.956,Z 359.578,A -85,B 0,C 180,E1 -6660.824,E2 -6660.824} C_VEL
LIN {X 0,Y 488.963,Z 359.577,A -85,B 0,C 180,E1 -6662.471,E2 -6662.471} C_VEL
LIN {X 0,Y 488.857,Z 359.59,A -85,B 0,C 180,E1 -6665.776,E2 -6665.776} C_VEL
LIN {X 0,Y 488.82,Z 359.597,A -85,B 0,C 180,E1 -6668.266,E2 -6668.266} C_VEL
LIN {X 0,Y 488.831,Z 359.596,A -85,B 0,C 180,E1 -6671.612,E2 -6671.612} C_VEL
LIN {X 0,Y 488.764,Z 359.603,A -85,B 0,C 180,E1 -6675,E2 -6675} C_VEL
LIN {X 0,Y 488.756,Z 359.604,A -85,B 0,C 180,E1 -6678.442,E2 -6678.442} C_VEL
LIN {X 0,Y 488.709,Z 359.609,A -85,B 0,C 180,E1 -6681.071,E2 -6681.071} C_VEL
LIN {X 0,Y 488.696,Z 359.612,A -85,B 0,C 180,E1 -6683.745,E2 -6683.745} C_VEL
LIN {X 0,Y 488.793,Z 359.602,A -85,B 0,C 180,E1 -6686.944,E2 -6686.944} C_VEL
LIN {X 0,Y 488.711,Z 359.611,A -85,B 0,C 180,E1 -6690.363,E2 -6690.363} C_VEL
LIN {X 0,Y 488.737,Z 359.609,A -85,B 0,C 180,E1 -6693.485,E2 -6693.485} C_VEL
LIN {X 0,Y 488.689,Z 359.61,A -85,B 0,C 180,E1 -6696.356,E2 -6696.356} C_VEL
LIN {X 0,Y 488.703,Z 359.609,A -85,B 0,C 180,E1 -6699.254,E2 -6699.254} C_VEL
LIN {X 0,Y 488.71,Z 359.61,A -85,B 0,C 180,E1 -6701.6,E2 -6701.6} C_VEL
LIN {X 0,Y 488.714,Z 359.609,A -85,B 0,C 180,E1 -6704.801,E2 -6704.801} C_VEL
LIN {X 0,Y 488.697,Z 359.609,A -85,B 0,C 180,E1 -6707.475,E2 -6707.475} C_VEL
LIN {X 0,Y 488.734,Z 359.604,A -85,B 0,C 180,E1 -6709.677,E2 -6709.677} C_VEL
LIN {X 0,Y 488.681,Z 359.612,A -85,B 0,C 180,E1 -6712.841,E2 -6712.841} C_VEL
LIN {X 0,Y 488.732,Z 359.606,A -85,B 0,C 180,E1 -6715.887,E2 -6715.887} C_VEL
LIN {X 0,Y 488.695,Z 359.612,A -85,B 0,C 180,E1 -6718.821,E2 -6718.821} C_VEL
LIN {X 0,Y 488.748,Z 359.604,A -85,B 0,C 180,E1 -6721.672,E2 -6721.672} C_VEL
LIN {X 0,Y 488.745,Z 359.604,A -85,B 0,C 180,E1 -6724.345,E2 -6724.345} C_VEL
LIN {X 0,Y 488.1,Z 359.687,A -85,B 0,C 180,E1 -6725.033,E2 -6725.033} C_VEL
LIN {X 0,Y 485.232,Z 360.043,A -85,B 0,C 180,E1 -6726.149,E2 -6726.149} C_VEL
LIN {X 0,Y 482.785,Z 360.349,A -85,B 0,C 180,E1 -6727.049,E2 -6727.049} C_VEL
LIN {X 0,Y 481.727,Z 360.478,A -85,B 0,C 180,E1 -6727.744,E2 -6727.744} C_VEL
LIN {X 0,Y 481.638,Z 360.489,A -85,B 0,C 180,E1 -6727.98,E2 -6727.98} C_VEL
LIN {X 0,Y 481.711,Z 360.484,A -85,B 0,C 180,E1 -6730.393,E2 -6730.393} C_VEL
LIN {X 0,Y 481.694,Z 360.482,A -85,B 0,C 180,E1 -6733.034,E2 -6733.034} C_VEL
LIN {X 0,Y 481.693,Z 360.486,A -85,B 0,C 180,E1 -6735.639,E2 -6735.639} C_VEL
LIN {X 0,Y 481.754,Z 360.476,A -85,B 0,C 180,E1 -6738.215,E2 -6738.215} C_VEL
LIN {X 0,Y 481.766,Z 360.473,A -85,B 0,C 180,E1 -6741.612,E2 -6741.612} C_VEL
LIN {X 0,Y 481.812,Z 360.469,A -85,B 0,C 180,E1 -6744.14,E2 -6744.14} C_VEL
LIN {X 0,Y 481.931,Z 360.455,A -85,B 0,C 180,E1 -6747.493,E2 -6747.493} C_VEL
LIN {X 0,Y 481.909,Z 360.456,A -85,B 0,C 180,E1 -6750.836,E2 -6750.836} C_VEL
LIN {X 0,Y 481.931,Z 360.452,A -85,B 0,C 180,E1 -6752.508,E2 -6752.508} C_VEL
LIN {X 0,Y 481.812,Z 360.469,A -85,B 0,C 180,E1 -6755.861,E2 -6755.861} C_VEL
LIN {X 0,Y 481.767,Z 360.476,A -85,B 0,C 180,E1 -6758.388,E2 -6758.388} C_VEL
LIN {X 0,Y 481.755,Z 360.477,A -85,B 0,C 180,E1 -6761.785,E2 -6761.785} C_VEL
LIN {X 0,Y 481.746,Z 360.477,A -85,B 0,C 180,E1 -6765.224,E2 -6765.224} C_VEL
LIN {X 0,Y 481.716,Z 360.482,A -85,B 0,C 180,E1 -6768.722,E2 -6768.722} C_VEL
LIN {X 0,Y 481.649,Z 360.488,A -85,B 0,C 180,E1 -6771.395,E2 -6771.395} C_VEL
LIN {X 0,Y 481.665,Z 360.486,A -85,B 0,C 180,E1 -6774.114,E2 -6774.114} C_VEL
LIN {X 0,Y 481.751,Z 360.478,A -85,B 0,C 180,E1 -6777.139,E2 -6777.139} C_VEL
LIN {X 0,Y 481.682,Z 360.484,A -85,B 0,C 180,E1 -6779.741,E2 -6779.741} C_VEL
LIN {X 0,Y 481.676,Z 360.485,A -85,B 0,C 180,E1 -6782.674,E2 -6782.674} C_VEL
LIN {X 0,Y 481.64,Z 360.49,A -85,B 0,C 180,E1 -6785.71,E2 -6785.71} C_VEL
LIN {X 0,Y 481.674,Z 360.488,A -85,B 0,C 180,E1 -6788.859,E2 -6788.859} C_VEL
LIN {X 0,Y 481.666,Z 360.489,A -85,B 0,C 180,E1 -6791.914,E2 -6791.914} C_VEL
LIN {X 0,Y 481.658,Z 360.486,A -85,B 0,C 180,E1 -6794.458,E2 -6794.458} C_VEL
LIN {X 0,Y 481.65,Z 360.487,A -85,B 0,C 180,E1 -6797.839,E2 -6797.839} C_VEL
LIN {X 0,Y 481.684,Z 360.487,A -85,B 0,C 180,E1 -6800.651,E2 -6800.651} C_VEL
LIN {X 0,Y 481.634,Z 360.491,A -85,B 0,C 180,E1 -6803.376,E2 -6803.376} C_VEL
LIN {X 0,Y 481.713,Z 360.479,A -85,B 0,C 180,E1 -6806.33,E2 -6806.33} C_VEL
LIN {X 0,Y 481.799,Z 360.549,A -85,B 0,C 180,E1 -6809.732,E2 -6809.732} C_VEL
LIN {X 0,Y 481.652,Z 366.973,A -85,B 0,C 180,E1 -6812.884,E2 -6812.884} C_VEL
LIN {X 0,Y 481.469,Z 373.185,A -85,B 0,C 180,E1 -6815.876,E2 -6815.876} C_VEL
LIN {X 0,Y 481.357,Z 379.979,A -85,B 0,C 180,E1 -6819.136,E2 -6819.136} C_VEL
LIN {X 0,Y 481.268,Z 386.387,A -85,B 0,C 180,E1 -6822.142,E2 -6822.142} C_VEL
LIN {X 0,Y 481.225,Z 392.011,A -85,B 0,C 180,E1 -6824.759,E2 -6824.759} C_VEL
LIN {X 0,Y 481.09,Z 399.488,A -85,B 0,C 180,E1 -6828.199,E2 -6828.199} C_VEL
LIN {X 0,Y 480.998,Z 405.916,A -85,B 0,C 180,E1 -6831.122,E2 -6831.122} C_VEL
LIN {X 0,Y 482.14,Z 414.559,A -85,B 0,C 180,E1 -6831.513,E2 -6831.513} C_VEL
LIN {X 0,Y 482.046,Z 423.679,A -85,B 0,C 180,E1 -6832.039,E2 -6832.039} C_VEL
LIN {X 0,Y 481.845,Z 432.733,A -85,B 0,C 180,E1 -6832.741,E2 -6832.741} C_VEL
LIN {X 0,Y 481.522,Z 440.315,A -85,B 0,C 180,E1 -6833.505,E2 -6833.505} C_VEL
LIN {X 0,Y 481.5,Z 446.814,A -85,B 0,C 180,E1 -6834.346,E2 -6834.346} C_VEL
LIN {X 0,Y 481.389,Z 453.049,A -85,B 0,C 180,E1 -6835.394,E2 -6835.394} C_VEL
LIN {X 0,Y 481.293,Z 456.863,A -85,B 0,C 180,E1 -6836.232,E2 -6836.232} C_VEL
LIN {X 0,Y 481.213,Z 459.823,A -85,B 0,C 180,E1 -6837.07,E2 -6837.07} C_VEL
LIN {X 0,Y 481.01,Z 461.022,A -85,B 0,C 180,E1 -6837.488,E2 -6837.488} C_VEL
LIN {X 0,Y 480.928,Z 462.839,A -85,B 0,C 180,E1 -6838.325,E2 -6838.325} C_VEL
LIN {X 0,Y 480.906,Z 463.955,A -85,B 0,C 180,E1 -6839.163,E2 -6839.163} C_VEL
LIN {X 0,Y 480.907,Z 464.401,A -85,B 0,C 180,E1 -6840,E2 -6840} C_VEL
LIN {X 0,Y 480.919,Z 464.182,A -85,B 0,C 180,E1 -6840.837,E2 -6840.837} C_VEL
LIN {X 0,Y 480.954,Z 463.295,A -85,B 0,C 180,E1 -6841.675,E2 -6841.675} C_VEL
LIN {X 0,Y 481.218,Z 460.647,A -85,B 0,C 180,E1 -6842.93,E2 -6842.93} C_VEL
LIN {X 0,Y 481.384,Z 457.942,A -85,B 0,C 180,E1 -6843.767,E2 -6843.767} C_VEL
LIN {X 0,Y 481.432,Z 453.398,A -85,B 0,C 180,E1 -6844.815,E2 -6844.815} C_VEL
LIN {X 0,Y 481.583,Z 447.237,A -85,B 0,C 180,E1 -6845.863,E2 -6845.863} C_VEL
LIN {X 0,Y 481.769,Z 440.835,A -85,B 0,C 180,E1 -6846.702,E2 -6846.702} C_VEL
LIN {X 0,Y 482.121,Z 432.042,A -85,B 0,C 180,E1 -6847.581,E2 -6847.581} C_VEL
LIN {X 0,Y 482.292,Z 422.878,A -85,B 0,C 180,E1 -6848.273,E2 -6848.273} C_VEL
LIN {X 0,Y 482.379,Z 414.578,A -85,B 0,C 180,E1 -6848.747,E2 -6848.747} C_VEL
LIN {X 0,Y 481.168,Z 407.387,A -85,B 0,C 180,E1 -6849.113,E2 -6849.113} C_VEL
LIN {X 0,Y 481.285,Z 401.409,A -85,B 0,C 180,E1 -6851.936,E2 -6851.936} C_VEL
LIN {X 0,Y 481.445,Z 393.896,A -85,B 0,C 180,E1 -6855.538,E2 -6855.538} C_VEL
LIN {X 0,Y 481.573,Z 387.374,A -85,B 0,C 180,E1 -6858.727,E2 -6858.727} C_VEL
LIN {X 0,Y 481.725,Z 381.999,A -85,B 0,C 180,E1 -6861.391,E2 -6861.391} C_VEL
LIN {X 0,Y 481.89,Z 376.607,A -85,B 0,C 180,E1 -6864.102,E2 -6864.102} C_VEL
LIN {X 0,Y 482.156,Z 370.509,A -85,B 0,C 180,E1 -6867.233,E2 -6867.233} C_VEL
LIN {X 0,Y 482.345,Z 365.925,A -85,B 0,C 180,E1 -6869.696,E2 -6869.696} C_VEL
LIN {X 0,Y 481.993,Z 362.379,A -85,B 0,C 180,E1 -6871.663,E2 -6871.663} C_VEL
LIN {X 0,Y 481.699,Z 360.486,A -85,B 0,C 180,E1 -6872.796,E2 -6872.796} C_VEL
LIN {X 0,Y 481.64,Z 360.493,A -85,B 0,C 180,E1 -6875.709,E2 -6875.709} C_VEL
LIN {X 0,Y 481.723,Z 360.482,A -85,B 0,C 180,E1 -6879.355,E2 -6879.355} C_VEL
LIN {X 0,Y 481.677,Z 360.488,A -85,B 0,C 180,E1 -6882.158,E2 -6882.158} C_VEL
LIN {X 0,Y 481.664,Z 360.49,A -85,B 0,C 180,E1 -6884.457,E2 -6884.457} C_VEL
LIN {X 0,Y 481.657,Z 360.491,A -85,B 0,C 180,E1 -6887.84,E2 -6887.84} C_VEL
LIN {X 0,Y 481.683,Z 360.488,A -85,B 0,C 180,E1 -6890.651,E2 -6890.651} C_VEL
LIN {X 0,Y 481.63,Z 360.495,A -85,B 0,C 180,E1 -6893.376,E2 -6893.376} C_VEL
LIN {X 0,Y 481.71,Z 360.504,A -85,B 0,C 180,E1 -6895.827,E2 -6895.827} C_VEL
LIN {X 0,Y 483.147,Z 366.621,A -85,B 0,C 180,E1 -6898.016,E2 -6898.016} C_VEL
LIN {X 0,Y 484.945,Z 374.782,A -85,B 0,C 180,E1 -6900.479,E2 -6900.479} C_VEL
LIN {X 0,Y 485.316,Z 378.46,A -85,B 0,C 180,E1 -6901.453,E2 -6901.453} C_VEL
LIN {X 0,Y 484.367,Z 388.183,A -85,B 0,C 180,E1 -6903.734,E2 -6903.734} C_VEL
LIN {X 0,Y 483.45,Z 401.239,A -85,B 0,C 180,E1 -6906.598,E2 -6906.598} C_VEL
LIN {X 0,Y 482.588,Z 417.778,A -85,B 0,C 180,E1 -6909.987,E2 -6909.987} C_VEL
LIN {X 0,Y 481.981,Z 434.61,A -85,B 0,C 180,E1 -6913.262,E2 -6913.262} C_VEL
LIN {X 0,Y 481.712,Z 445.607,A -85,B 0,C 180,E1 -6915.342,E2 -6915.342} C_VEL
LIN {X 0,Y 483.172,Z 459.431,A -85,B 0,C 180,E1 -6915.697,E2 -6915.697} C_VEL
LIN {X 0,Y 483.267,Z 468.555,A -85,B 0,C 180,E1 -6916.009,E2 -6916.009} C_VEL
LIN {X 0,Y 482.943,Z 480.201,A -85,B 0,C 180,E1 -6916.536,E2 -6916.536} C_VEL
LIN {X 0,Y 482.564,Z 492.547,A -85,B 0,C 180,E1 -6917.274,E2 -6917.274} C_VEL
LIN {X 0,Y 482.223,Z 503.691,A -85,B 0,C 180,E1 -6918.134,E2 -6918.134} C_VEL
LIN {X 0,Y 481.856,Z 513.48,A -85,B 0,C 180,E1 -6919.07,E2 -6919.07} C_VEL
LIN {X 0,Y 481.5,Z 522.518,A -85,B 0,C 180,E1 -6920.125,E2 -6920.125} C_VEL
LIN {X 0,Y 481.284,Z 529.967,A -85,B 0,C 180,E1 -6921.18,E2 -6921.18} C_VEL
LIN {X 0,Y 481.118,Z 537.268,A -85,B 0,C 180,E1 -6922.445,E2 -6922.445} C_VEL
LIN {X 0,Y 480.986,Z 543.279,A -85,B 0,C 180,E1 -6923.764,E2 -6923.764} C_VEL
LIN {X 0,Y 480.912,Z 547.606,A -85,B 0,C 180,E1 -6924.969,E2 -6924.969} C_VEL
LIN {X 0,Y 481,Z 550.017,A -85,B 0,C 180,E1 -6925.81,E2 -6925.81} C_VEL
LIN {X 0,Y 480.964,Z 551.972,A -85,B 0,C 180,E1 -6926.649,E2 -6926.649} C_VEL
LIN {X 0,Y 480.935,Z 553.445,A -85,B 0,C 180,E1 -6927.487,E2 -6927.487} C_VEL
LIN {X 0,Y 480.812,Z 555.132,A -85,B 0,C 180,E1 -6929.162,E2 -6929.162} C_VEL
LIN {X 0,Y 480.811,Z 555.374,A -85,B 0,C 180,E1 -6930,E2 -6930} C_VEL
LIN {X 0,Y 480.81,Z 555.162,A -85,B 0,C 180,E1 -6930.837,E2 -6930.837} C_VEL
LIN {X 0,Y 480.935,Z 553.555,A -85,B 0,C 180,E1 -6932.512,E2 -6932.512} C_VEL
LIN {X 0,Y 480.963,Z 552.111,A -85,B 0,C 180,E1 -6933.351,E2 -6933.351} C_VEL
LIN {X 0,Y 480.892,Z 549.085,A -85,B 0,C 180,E1 -6934.61,E2 -6934.61} C_VEL
LIN {X 0,Y 481.018,Z 544.988,A -85,B 0,C 180,E1 -6935.87,E2 -6935.87} C_VEL
LIN {X 0,Y 481.111,Z 538.655,A -85,B 0,C 180,E1 -6937.343,E2 -6937.343} C_VEL
LIN {X 0,Y 481.284,Z 531.741,A -85,B 0,C 180,E1 -6938.608,E2 -6938.608} C_VEL
LIN {X 0,Y 481.473,Z 524.66,A -85,B 0,C 180,E1 -6939.664,E2 -6939.664} C_VEL
LIN {X 0,Y 481.789,Z 516.104,A -85,B 0,C 180,E1 -6940.719,E2 -6940.719} C_VEL
LIN {X 0,Y 482.151,Z 505.49,A -85,B 0,C 180,E1 -6941.775,E2 -6941.775} C_VEL
LIN {X 0,Y 482.502,Z 494.963,A -85,B 0,C 180,E1 -6942.62,E2 -6942.62} C_VEL
LIN {X 0,Y 482.903,Z 483.329,A -85,B 0,C 180,E1 -6943.358,E2 -6943.358} C_VEL
LIN {X 0,Y 483.246,Z 471.224,A -85,B 0,C 180,E1 -6943.938,E2 -6943.938} C_VEL
LIN {X 0,Y 483.348,Z 460.323,A -85,B 0,C 180,E1 -6944.324,E2 -6944.324} C_VEL
LIN {X 0,Y 482.023,Z 448.697,A -85,B 0,C 180,E1 -6944.634,E2 -6944.634} C_VEL
LIN {X 0,Y 481.794,Z 446.025,A -85,B 0,C 180,E1 -6944.709,E2 -6944.709} C_VEL
LIN {X 0,Y 482.327,Z 427.622,A -85,B 0,C 180,E1 -6948.257,E2 -6948.257} C_VEL
LIN {X 0,Y 483.021,Z 411.833,A -85,B 0,C 180,E1 -6951.376,E2 -6951.376} C_VEL
LIN {X 0,Y 483.897,Z 394.276,A -85,B 0,C 180,E1 -6954.91,E2 -6954.91} C_VEL
LIN {X 0,Y 484.866,Z 378.702,A -85,B 0,C 180,E1 -6958.138,E2 -6958.138} C_VEL
LIN {X 0,Y 484.858,Z 375.548,A -85,B 0,C 180,E1 -6958.813,E2 -6958.813} C_VEL
LIN {X 0,Y 482.776,Z 365.425,A -85,B 0,C 180,E1 -6961.178,E2 -6961.178} C_VEL
LIN {X 0,Y 481.668,Z 360.489,A -85,B 0,C 180,E1 -6962.393,E2 -6962.393} C_VEL
LIN {X 0,Y 481.664,Z 360.49,A -85,B 0,C 180,E1 -6965.204,E2 -6965.204} C_VEL
LIN {X 0,Y 481.672,Z 360.486,A -85,B 0,C 180,E1 -6968.859,E2 -6968.859} C_VEL
LIN {X 0,Y 481.664,Z 360.49,A -85,B 0,C 180,E1 -6971.914,E2 -6971.914} C_VEL
LIN {X 0,Y 481.662,Z 360.487,A -85,B 0,C 180,E1 -6974.457,E2 -6974.457} C_VEL
LIN {X 0,Y 481.655,Z 360.487,A -85,B 0,C 180,E1 -6977.84,E2 -6977.84} C_VEL
LIN {X 0,Y 481.682,Z 360.483,A -85,B 0,C 180,E1 -6980.651,E2 -6980.651} C_VEL
LIN {X 0,Y 481.633,Z 360.492,A -85,B 0,C 180,E1 -6983.375,E2 -6983.375} C_VEL
LIN {X 0,Y 481.711,Z 360.481,A -85,B 0,C 180,E1 -6986.33,E2 -6986.33} C_VEL
LIN {X 0,Y 481.652,Z 360.487,A -85,B 0,C 180,E1 -6989.417,E2 -6989.417} C_VEL
LIN {X 0,Y 481.702,Z 360.483,A -85,B 0,C 180,E1 -6992.168,E2 -6992.168} C_VEL
LIN {X 0,Y 481.718,Z 360.481,A -85,B 0,C 180,E1 -6994.97,E2 -6994.97} C_VEL
LIN {X 0,Y 481.65,Z 360.488,A -85,B 0,C 180,E1 -6997.705,E2 -6997.705} C_VEL
LIN {X 0,Y 481.709,Z 360.482,A -85,B 0,C 180,E1 -7000.393,E2 -7000.393} C_VEL
LIN {X 0,Y 481.693,Z 360.481,A -85,B 0,C 180,E1 -7003.034,E2 -7003.034} C_VEL
LIN {X 0,Y 481.696,Z 360.484,A -85,B 0,C 180,E1 -7005.639,E2 -7005.639} C_VEL
LIN {X 0,Y 481.753,Z 360.478,A -85,B 0,C 180,E1 -7008.215,E2 -7008.215} C_VEL
LIN {X 0,Y 481.764,Z 360.476,A -85,B 0,C 180,E1 -7011.612,E2 -7011.612} C_VEL
LIN {X 0,Y 481.818,Z 360.466,A -85,B 0,C 180,E1 -7014.14,E2 -7014.14} C_VEL
LIN {X 0,Y 481.93,Z 360.454,A -85,B 0,C 180,E1 -7017.493,E2 -7017.493} C_VEL
LIN {X 0,Y 481.907,Z 360.456,A -85,B 0,C 180,E1 -7020.836,E2 -7020.836} C_VEL
LIN {X 0,Y 481.93,Z 360.453,A -85,B 0,C 180,E1 -7022.507,E2 -7022.507} C_VEL
LIN {X 0,Y 481.818,Z 360.466,A -85,B 0,C 180,E1 -7025.86,E2 -7025.86} C_VEL
LIN {X 0,Y 481.765,Z 360.475,A -85,B 0,C 180,E1 -7028.388,E2 -7028.388} C_VEL
LIN {X 0,Y 481.797,Z 360.473,A -85,B 0,C 180,E1 -7031.784,E2 -7031.784} C_VEL
LIN {X 0,Y 481.744,Z 360.48,A -85,B 0,C 180,E1 -7035.224,E2 -7035.224} C_VEL
LIN {X 0,Y 481.714,Z 360.483,A -85,B 0,C 180,E1 -7038.722,E2 -7038.722} C_VEL
LIN {X 0,Y 481.649,Z 360.489,A -85,B 0,C 180,E1 -7041.395,E2 -7041.395} C_VEL
LIN {X 0,Y 481.679,Z 360.484,A -85,B 0,C 180,E1 -7044.113,E2 -7044.113} C_VEL
LIN {X 0,Y 481.748,Z 360.478,A -85,B 0,C 180,E1 -7047.139,E2 -7047.139} C_VEL
LIN {X 0,Y 481.68,Z 360.485,A -85,B 0,C 180,E1 -7049.741,E2 -7049.741} C_VEL
LIN {X 0,Y 481.674,Z 360.485,A -85,B 0,C 180,E1 -7052.674,E2 -7052.674} C_VEL
LIN {X 0,Y 481.643,Z 360.489,A -85,B 0,C 180,E1 -7055.709,E2 -7055.709} C_VEL
LIN {X 0,Y 481.673,Z 360.488,A -85,B 0,C 180,E1 -7058.859,E2 -7058.859} C_VEL
LIN {X 0,Y 481.655,Z 360.489,A -85,B 0,C 180,E1 -7061.913,E2 -7061.913} C_VEL
LIN {X 0,Y 481.661,Z 360.487,A -85,B 0,C 180,E1 -7064.457,E2 -7064.457} C_VEL
LIN {X 0,Y 481.655,Z 360.485,A -85,B 0,C 180,E1 -7067.84,E2 -7067.84} C_VEL
LIN {X 0,Y 481.682,Z 360.486,A -85,B 0,C 180,E1 -7070.651,E2 -7070.651} C_VEL
LIN {X 0,Y 481.629,Z 360.493,A -85,B 0,C 180,E1 -7073.376,E2 -7073.376} C_VEL
LIN {X 0,Y 481.711,Z 360.48,A -85,B 0,C 180,E1 -7076.33,E2 -7076.33} C_VEL
LIN {X 0,Y 481.653,Z 360.485,A -85,B 0,C 180,E1 -7079.418,E2 -7079.418} C_VEL
LIN {X 0,Y 481.703,Z 360.485,A -85,B 0,C 180,E1 -7082.168,E2 -7082.168} C_VEL
LIN {X 0,Y 481.72,Z 360.481,A -85,B 0,C 180,E1 -7084.97,E2 -7084.97} C_VEL
LIN {X 0,Y 481.638,Z 360.489,A -85,B 0,C 180,E1 -7087.98,E2 -7087.98} C_VEL
LIN {X 0,Y 480.971,Z 360.576,A -85,B 0,C 180,E1 -7088.678,E2 -7088.678} C_VEL
LIN {X 0,Y 478.145,Z 360.924,A -85,B 0,C 180,E1 -7089.812,E2 -7089.812} C_VEL
LIN {X 0,Y 475.761,Z 361.222,A -85,B 0,C 180,E1 -7090.727,E2 -7090.727} C_VEL
LIN {X 0,Y 474.74,Z 361.347,A -85,B 0,C 180,E1 -7091.433,E2 -7091.433} C_VEL
LIN {X 0,Y 474.658,Z 361.358,A -85,B 0,C 180,E1 -7091.671,E2 -7091.671} C_VEL
LIN {X 0,Y 474.703,Z 361.353,A -85,B 0,C 180,E1 -7094.545,E2 -7094.545} C_VEL
LIN {X 0,Y 474.708,Z 361.353,A -85,B 0,C 180,E1 -7098.038,E2 -7098.038} C_VEL
LIN {X 0,Y 474.731,Z 361.348,A -85,B 0,C 180,E1 -7101.487,E2 -7101.487} C_VEL
LIN {X 0,Y 474.774,Z 361.346,A -85,B 0,C 180,E1 -7104.052,E2 -7104.052} C_VEL
LIN {X 0,Y 474.897,Z 361.331,A -85,B 0,C 180,E1 -7107.456,E2 -7107.456} C_VEL
LIN {X 0,Y 474.916,Z 361.328,A -85,B 0,C 180,E1 -7110,E2 -7110} C_VEL
LIN {X 0,Y 474.897,Z 361.328,A -85,B 0,C 180,E1 -7112.545,E2 -7112.545} C_VEL
LIN {X 0,Y 474.774,Z 361.345,A -85,B 0,C 180,E1 -7115.948,E2 -7115.948} C_VEL
LIN {X 0,Y 474.732,Z 361.352,A -85,B 0,C 180,E1 -7118.514,E2 -7118.514} C_VEL
LIN {X 0,Y 474.709,Z 361.357,A -85,B 0,C 180,E1 -7121.963,E2 -7121.963} C_VEL
LIN {X 0,Y 474.704,Z 361.357,A -85,B 0,C 180,E1 -7125.456,E2 -7125.456} C_VEL
LIN {X 0,Y 474.668,Z 361.36,A -85,B 0,C 180,E1 -7129.01,E2 -7129.01} C_VEL
LIN {X 0,Y 474.592,Z 361.369,A -85,B 0,C 180,E1 -7131.729,E2 -7131.729} C_VEL
LIN {X 0,Y 474.645,Z 361.358,A -85,B 0,C 180,E1 -7134.494,E2 -7134.494} C_VEL
LIN {X 0,Y 474.703,Z 361.357,A -85,B 0,C 180,E1 -7137.339,E2 -7137.339} C_VEL
LIN {X 0,Y 474.608,Z 361.367,A -85,B 0,C 180,E1 -7140.81,E2 -7140.81} C_VEL
LIN {X 0,Y 474.64,Z 361.362,A -85,B 0,C 180,E1 -7143.984,E2 -7143.984} C_VEL
LIN {X 0,Y 474.575,Z 361.37,A -85,B 0,C 180,E1 -7146.899,E2 -7146.899} C_VEL
LIN {X 0,Y 474.631,Z 361.362,A -85,B 0,C 180,E1 -7149.648,E2 -7149.648} C_VEL
LIN {X 0,Y 474.638,Z 361.361,A -85,B 0,C 180,E1 -7152.932,E2 -7152.932} C_VEL
LIN {X 0,Y 474.609,Z 361.364,A -85,B 0,C 180,E1 -7155.895,E2 -7155.895} C_VEL
LIN {X 0,Y 474.63,Z 361.365,A -85,B 0,C 180,E1 -7159.041,E2 -7159.041} C_VEL
LIN {X 0,Y 474.614,Z 361.366,A -85,B 0,C 180,E1 -7161.704,E2 -7161.704} C_VEL
LIN {X 0,Y 474.633,Z 361.362,A -85,B 0,C 180,E1 -7164.726,E2 -7164.726} C_VEL
LIN {X 0,Y 474.64,Z 361.361,A -85,B 0,C 180,E1 -7167.788,E2 -7167.788} C_VEL
LIN {X 0,Y 474.739,Z 361.423,A -85,B 0,C 180,E1 -7169.68,E2 -7169.68} C_VEL
LIN {X 0,Y 474.62,Z 367.487,A -85,B 0,C 180,E1 -7172.681,E2 -7172.681} C_VEL
LIN {X 0,Y 474.448,Z 373.262,A -85,B 0,C 180,E1 -7175.495,E2 -7175.495} C_VEL
LIN {X 0,Y 474.321,Z 378.985,A -85,B 0,C 180,E1 -7178.258,E2 -7178.258} C_VEL
LIN {X 0,Y 474.237,Z 385.828,A -85,B 0,C 180,E1 -7181.524,E2 -7181.524} C_VEL
LIN {X 0,Y 474.186,Z 392.225,A -85,B 0,C 180,E1 -7184.527,E2 -7184.527} C_VEL
LIN {X 0,Y 474.031,Z 399.94,A -85,B 0,C 180,E1 -7188.104,E2 -7188.104} C_VEL
LIN {X 0,Y 473.935,Z 406.187,A -85,B 0,C 180,E1 -7190.962,E2 -7190.962} C_VEL
LIN {X 0,Y 475.153,Z 415.227,A -85,B 0,C 180,E1 -7191.387,E2 -7191.387} C_VEL
LIN {X 0,Y 475.061,Z 424.261,A -85,B 0,C 180,E1 -7191.921,E2 -7191.921} C_VEL
LIN {X 0,Y 474.855,Z 432.696,A -85,B 0,C 180,E1 -7192.58,E2 -7192.58} C_VEL
LIN {X 0,Y 474.504,Z 440.864,A -85,B 0,C 180,E1 -7193.409,E2 -7193.409} C_VEL
LIN {X 0,Y 474.484,Z 447.375,A -85,B 0,C 180,E1 -7194.262,E2 -7194.262} C_VEL
LIN {X 0,Y 474.362,Z 453.631,A -85,B 0,C 180,E1 -7195.326,E2 -7195.326} C_VEL
LIN {X 0,Y 474.144,Z 459.064,A -85,B 0,C 180,E1 -7196.601,E2 -7196.601} C_VEL
LIN {X 0,Y 473.954,Z 461.656,A -85,B 0,C 180,E1 -7197.45,E2 -7197.45} C_VEL
LIN {X 0,Y 473.861,Z 463.491,A -85,B 0,C 180,E1 -7198.3,E2 -7198.3} C_VEL
LIN {X 0,Y 473.839,Z 464.623,A -85,B 0,C 180,E1 -7199.15,E2 -7199.15} C_VEL
LIN {X 0,Y 473.84,Z 465.083,A -85,B 0,C 180,E1 -7200,E2 -7200} C_VEL
LIN {X 0,Y 473.854,Z 464.877,A -85,B 0,C 180,E1 -7200.85,E2 -7200.85} C_VEL
LIN {X 0,Y 473.893,Z 464.002,A -85,B 0,C 180,E1 -7201.7,E2 -7201.7} C_VEL
LIN {X 0,Y 474.179,Z 461.369,A -85,B 0,C 180,E1 -7202.974,E2 -7202.974} C_VEL
LIN {X 0,Y 474.355,Z 458.676,A -85,B 0,C 180,E1 -7203.823,E2 -7203.823} C_VEL
LIN {X 0,Y 474.412,Z 454.152,A -85,B 0,C 180,E1 -7204.886,E2 -7204.886} C_VEL
LIN {X 0,Y 474.581,Z 448.043,A -85,B 0,C 180,E1 -7205.95,E2 -7205.95} C_VEL
LIN {X 0,Y 474.772,Z 441.712,A -85,B 0,C 180,E1 -7206.801,E2 -7206.801} C_VEL
LIN {X 0,Y 475.155,Z 433.068,A -85,B 0,C 180,E1 -7207.693,E2 -7207.693} C_VEL
LIN {X 0,Y 475.364,Z 424.124,A -85,B 0,C 180,E1 -7208.395,E2 -7208.395} C_VEL
LIN {X 0,Y 475.43,Z 415.099,A -85,B 0,C 180,E1 -7208.929,E2 -7208.929} C_VEL
LIN {X 0,Y 474.136,Z 407.844,A -85,B 0,C 180,E1 -7209.303,E2 -7209.303} C_VEL
LIN {X 0,Y 474.245,Z 402.153,A -85,B 0,C 180,E1 -7212.018,E2 -7212.018} C_VEL
LIN {X 0,Y 474.411,Z 394.687,A -85,B 0,C 180,E1 -7215.651,E2 -7215.651} C_VEL
LIN {X 0,Y 474.569,Z 387.909,A -85,B 0,C 180,E1 -7219.014,E2 -7219.014} C_VEL
LIN {X 0,Y 474.73,Z 382.555,A -85,B 0,C 180,E1 -7221.722,E2 -7221.722} C_VEL
LIN {X 0,Y 474.925,Z 377.191,A -85,B 0,C 180,E1 -7224.478,E2 -7224.478} C_VEL
LIN {X 0,Y 475.215,Z 371.577,A -85,B 0,C 180,E1 -7227.458,E2 -7227.458} C_VEL
LIN {X 0,Y 475.406,Z 368.21,A -85,B 0,C 180,E1 -7229.283,E2 -7229.283} C_VEL
LIN {X 0,Y 475.211,Z 364.841,A -85,B 0,C 180,E1 -7231.173,E2 -7231.173} C_VEL
LIN {X 0,Y 474.668,Z 361.362,A -85,B 0,C 180,E1 -7233.343,E2 -7233.343} C_VEL
LIN {X 0,Y 474.592,Z 361.371,A -85,B 0,C 180,E1 -7236.323,E2 -7236.323} C_VEL
LIN {X 0,Y 474.659,Z 361.362,A -85,B 0,C 180,E1 -7239.652,E2 -7239.652} C_VEL
LIN {X 0,Y 474.655,Z 361.363,A -85,B 0,C 180,E1 -7242.93,E2 -7242.93} C_VEL
LIN {X 0,Y 474.618,Z 361.366,A -85,B 0,C 180,E1 -7245.896,E2 -7245.896} C_VEL
LIN {X 0,Y 474.635,Z 361.365,A -85,B 0,C 180,E1 -7249.04,E2 -7249.04} C_VEL
LIN {X 0,Y 474.612,Z 361.368,A -85,B 0,C 180,E1 -7251.704,E2 -7251.704} C_VEL
LIN {X 0,Y 474.67,Z 361.462,A -85,B 0,C 180,E1 -7255.183,E2 -7255.183} C_VEL
LIN {X 0,Y 476.017,Z 366.938,A -85,B 0,C 180,E1 -7257.305,E2 -7257.305} C_VEL
LIN {X 0,Y 477.938,Z 375.906,A -85,B 0,C 180,E1 -7260.18,E2 -7260.18} C_VEL
LIN {X 0,Y 478.42,Z 378.892,A -85,B 0,C 180,E1 -7261.002,E2 -7261.002} C_VEL
LIN {X 0,Y 478.29,Z 382.545,A -85,B 0,C 180,E1 -7261.952,E2 -7261.952} C_VEL
LIN {X 0,Y 476.885,Z 396.342,A -85,B 0,C 180,E1 -7265.164,E2 -7265.164} C_VEL
LIN {X 0,Y 476.003,Z 409.947,A -85,B 0,C 180,E1 -7268.111,E2 -7268.111} C_VEL
LIN {X 0,Y 475.307,Z 424.752,A -85,B 0,C 180,E1 -7271.142,E2 -7271.142} C_VEL
LIN {X 0,Y 474.784,Z 440.273,A -85,B 0,C 180,E1 -7274.189,E2 -7274.189} C_VEL
LIN {X 0,Y 474.647,Z 445.3,A -85,B 0,C 180,E1 -7275.16,E2 -7275.16} C_VEL
LIN {X 0,Y 476.03,Z 458.681,A -85,B 0,C 180,E1 -7275.505,E2 -7275.505} C_VEL
LIN {X 0,Y 476.337,Z 464.183,A -85,B 0,C 180,E1 -7275.692,E2 -7275.692} C_VEL
LIN {X 0,Y 476.028,Z 476.922,A -85,B 0,C 180,E1 -7276.227,E2 -7276.227} C_VEL
LIN {X 0,Y 475.678,Z 488.264,A -85,B 0,C 180,E1 -7276.87,E2 -7276.87} C_VEL
LIN {X 0,Y 475.335,Z 500.01,A -85,B 0,C 180,E1 -7277.73,E2 -7277.73} C_VEL
LIN {X 0,Y 474.847,Z 510.543,A -85,B 0,C 180,E1 -7278.69,E2 -7278.69} C_VEL
LIN {X 0,Y 474.509,Z 519.996,A -85,B 0,C 180,E1 -7279.762,E2 -7279.762} C_VEL
LIN {X 0,Y 474.227,Z 529.154,A -85,B 0,C 180,E1 -7281.048,E2 -7281.048} C_VEL
LIN {X 0,Y 474.043,Z 536.5,A -85,B 0,C 180,E1 -7282.332,E2 -7282.332} C_VEL
LIN {X 0,Y 473.895,Z 542.999,A -85,B 0,C 180,E1 -7283.787,E2 -7283.787} C_VEL
LIN {X 0,Y 473.851,Z 546.898,A -85,B 0,C 180,E1 -7284.894,E2 -7284.894} C_VEL
LIN {X 0,Y 473.896,Z 549.316,A -85,B 0,C 180,E1 -7285.747,E2 -7285.747} C_VEL
LIN {X 0,Y 473.892,Z 551.283,A -85,B 0,C 180,E1 -7286.599,E2 -7286.599} C_VEL
LIN {X 0,Y 473.876,Z 552.77,A -85,B 0,C 180,E1 -7287.45,E2 -7287.45} C_VEL
LIN {X 0,Y 473.742,Z 554.469,A -85,B 0,C 180,E1 -7289.15,E2 -7289.15} C_VEL
LIN {X 0,Y 473.742,Z 554.715,A -85,B 0,C 180,E1 -7290,E2 -7290} C_VEL
LIN {X 0,Y 473.739,Z 554.506,A -85,B 0,C 180,E1 -7290.85,E2 -7290.85} C_VEL
LIN {X 0,Y 473.876,Z 552.9,A -85,B 0,C 180,E1 -7292.55,E2 -7292.55} C_VEL
LIN {X 0,Y 473.889,Z 551.447,A -85,B 0,C 180,E1 -7293.401,E2 -7293.401} C_VEL
LIN {X 0,Y 473.808,Z 548.412,A -85,B 0,C 180,E1 -7294.679,E2 -7294.679} C_VEL
LIN {X 0,Y 473.911,Z 544.298,A -85,B 0,C 180,E1 -7295.958,E2 -7295.958} C_VEL
LIN {X 0,Y 474.022,Z 537.949,A -85,B 0,C 180,E1 -7297.454,E2 -7297.454} C_VEL
LIN {X 0,Y 474.184,Z 531.007,A -85,B 0,C 180,E1 -7298.738,E2 -7298.738} C_VEL
LIN {X 0,Y 474.413,Z 523.897,A -85,B 0,C 180,E1 -7299.809,E2 -7299.809} C_VEL
LIN {X 0,Y 474.746,Z 515.277,A -85,B 0,C 180,E1 -7300.88,E2 -7300.88} C_VEL
LIN {X 0,Y 475.163,Z 504.608,A -85,B 0,C 180,E1 -7301.951,E2 -7301.951} C_VEL
LIN {X 0,Y 475.533,Z 493.998,A -85,B 0,C 180,E1 -7302.808,E2 -7302.808} C_VEL
LIN {X 0,Y 475.941,Z 482.165,A -85,B 0,C 180,E1 -7303.557,E2 -7303.557} C_VEL
LIN {X 0,Y 476.336,Z 469.86,A -85,B 0,C 180,E1 -7304.144,E2 -7304.144} C_VEL
LIN {X 0,Y 476.299,Z 460.365,A -85,B 0,C 180,E1 -7304.486,E2 -7304.486} C_VEL
LIN {X 0,Y 475.071,Z 449.017,A -85,B 0,C 180,E1 -7304.798,E2 -7304.798} C_VEL
LIN {X 0,Y 474.722,Z 445.819,A -85,B 0,C 180,E1 -7304.878,E2 -7304.878} C_VEL
LIN {X 0,Y 475.264,Z 429.506,A -85,B 0,C 180,E1 -7308.092,E2 -7308.092} C_VEL
LIN {X 0,Y 475.928,Z 414.206,A -85,B 0,C 180,E1 -7311.153,E2 -7311.153} C_VEL
LIN {X 0,Y 476.751,Z 398.401,A -85,B 0,C 180,E1 -7314.378,E2 -7314.378} C_VEL
LIN {X 0,Y 477.873,Z 381.453,A -85,B 0,C 180,E1 -7317.953,E2 -7317.953} C_VEL
LIN {X 0,Y 478.026,Z 377.616,A -85,B 0,C 180,E1 -7318.783,E2 -7318.783} C_VEL
LIN {X 0,Y 476.188,Z 368.377,A -85,B 0,C 180,E1 -7320.959,E2 -7320.959} C_VEL
LIN {X 0,Y 474.647,Z 361.363,A -85,B 0,C 180,E1 -7322.678,E2 -7322.678} C_VEL
LIN {X 0,Y 474.616,Z 361.367,A -85,B 0,C 180,E1 -7325.469,E2 -7325.469} C_VEL
LIN {X 0,Y 474.613,Z 361.367,A -85,B 0,C 180,E1 -7328.457,E2 -7328.457} C_VEL
LIN {X 0,Y 474.634,Z 361.361,A -85,B 0,C 180,E1 -7330.96,E2 -7330.96} C_VEL
LIN {X 0,Y 474.616,Z 361.365,A -85,B 0,C 180,E1 -7334.104,E2 -7334.104} C_VEL
LIN {X 0,Y 474.637,Z 361.363,A -85,B 0,C 180,E1 -7337.068,E2 -7337.068} C_VEL
LIN {X 0,Y 474.646,Z 361.361,A -85,B 0,C 180,E1 -7340.454,E2 -7340.454} C_VEL
LIN {X 0,Y 474.594,Z 361.37,A -85,B 0,C 180,E1 -7343.677,E2 -7343.677} C_VEL
LIN {X 0,Y 474.644,Z 361.363,A -85,B 0,C 180,E1 -7346.78,E2 -7346.78} C_VEL
LIN {X 0,Y 474.606,Z 361.366,A -85,B 0,C 180,E1 -7349.77,E2 -7349.77} C_VEL
LIN {X 0,Y 474.698,Z 361.353,A -85,B 0,C 180,E1 -7352.68,E2 -7352.68} C_VEL
LIN {X 0,Y 474.658,Z 361.362,A -85,B 0,C 180,E1 -7355.507,E2 -7355.507} C_VEL
LIN {X 0,Y 474.672,Z 361.357,A -85,B 0,C 180,E1 -7359.185,E2 -7359.185} C_VEL
LIN {X 0,Y 474.658,Z 361.363,A -85,B 0,C 180,E1 -7361.884,E2 -7361.884} C_VEL
LIN {X 0,Y 474.702,Z 361.353,A -85,B 0,C 180,E1 -7364.544,E2 -7364.544} C_VEL
LIN {X 0,Y 474.706,Z 361.354,A -85,B 0,C 180,E1 -7368.038,E2 -7368.038} C_VEL
LIN {X 0,Y 474.73,Z 361.351,A -85,B 0,C 180,E1 -7371.486,E2 -7371.486} C_VEL
LIN {X 0,Y 474.78,Z 361.343,A -85,B 0,C 180,E1 -7374.052,E2 -7374.052} C_VEL
LIN {X 0,Y 474.896,Z 361.33,A -85,B 0,C 180,E1 -7377.455,E2 -7377.455} C_VEL
LIN {X 0,Y 474.914,Z 361.33,A -85,B 0,C 180,E1 -7380,E2 -7380} C_VEL
LIN {X 0,Y 474.896,Z 361.329,A -85,B 0,C 180,E1 -7382.545,E2 -7382.545} C_VEL
LIN {X 0,Y 474.781,Z 361.343,A -85,B 0,C 180,E1 -7385.948,E2 -7385.948} C_VEL
LIN {X 0,Y 474.73,Z 361.352,A -85,B 0,C 180,E1 -7388.514,E2 -7388.514} C_VEL
LIN {X 0,Y 474.741,Z 361.351,A -85,B 0,C 180,E1 -7391.962,E2 -7391.962} C_VEL
LIN {X 0,Y 474.682,Z 361.355,A -85,B 0,C 180,E1 -7395.768,E2 -7395.768} C_VEL
LIN {X 0,Y 474.667,Z 361.36,A -85,B 0,C 180,E1 -7399.01,E2 -7399.01} C_VEL
LIN {X 0,Y 474.593,Z 361.37,A -85,B 0,C 180,E1 -7401.729,E2 -7401.729} C_VEL
LIN {X 0,Y 474.661,Z 361.358,A -85,B 0,C 180,E1 -7404.493,E2 -7404.493} C_VEL
LIN {X 0,Y 474.682,Z 361.357,A -85,B 0,C 180,E1 -7407.334,E2 -7407.334} C_VEL
LIN {X 0,Y 474.607,Z 361.367,A -85,B 0,C 180,E1 -7410.23,E2 -7410.23} C_VEL
LIN {X 0,Y 474.644,Z 361.362,A -85,B 0,C 180,E1 -7413.22,E2 -7413.22} C_VEL
LIN {X 0,Y 474.593,Z 361.366,A -85,B 0,C 180,E1 -7416.323,E2 -7416.323} C_VEL
LIN {X 0,Y 474.629,Z 361.362,A -85,B 0,C 180,E1 -7419.648,E2 -7419.648} C_VEL
LIN {X 0,Y 474.616,Z 361.365,A -85,B 0,C 180,E1 -7422.934,E2 -7422.934} C_VEL
LIN {X 0,Y 474.617,Z 361.364,A -85,B 0,C 180,E1 -7425.896,E2 -7425.896} C_VEL
LIN {X 0,Y 474.634,Z 361.362,A -85,B 0,C 180,E1 -7429.04,E2 -7429.04} C_VEL
LIN {X 0,Y 474.611,Z 361.366,A -85,B 0,C 180,E1 -7431.704,E2 -7431.704} C_VEL
LIN {X 0,Y 474.626,Z 361.364,A -85,B 0,C 180,E1 -7434.726,E2 -7434.726} C_VEL
LIN {X 0,Y 474.638,Z 361.36,A -85,B 0,C 180,E1 -7437.788,E2 -7437.788} C_VEL
LIN {X 0,Y 474.626,Z 361.363,A -85,B 0,C 180,E1 -7440.885,E2 -7440.885} C_VEL
LIN {X 0,Y 474.663,Z 361.36,A -85,B 0,C 180,E1 -7443.629,E2 -7443.629} C_VEL
LIN {X 0,Y 474.638,Z 361.363,A -85,B 0,C 180,E1 -7446.642,E2 -7446.642} C_VEL
LIN {X 0,Y 474.66,Z 361.36,A -85,B 0,C 180,E1 -7450.09,E2 -7450.09} C_VEL
LIN {X 0,Y 474.658,Z 361.358,A -85,B 0,C 180,E1 -7451.671,E2 -7451.671} C_VEL
LIN {X 0,Y 473.996,Z 361.446,A -85,B 0,C 180,E1 -7452.381,E2 -7452.381} C_VEL
LIN {X 0,Y 471.145,Z 361.803,A -85,B 0,C 180,E1 -7453.532,E2 -7453.532} C_VEL
LIN {X 0,Y 468.729,Z 362.102,A -85,B 0,C 180,E1 -7454.461,E2 -7454.461} C_VEL
LIN {X 0,Y 467.687,Z 362.229,A -85,B 0,C 180,E1 -7455.178,E2 -7455.178} C_VEL
LIN {X 0,Y 467.6,Z 362.238,A -85,B 0,C 180,E1 -7455.421,E2 -7455.421} C_VEL
LIN {X 0,Y 467.656,Z 362.233,A -85,B 0,C 180,E1 -7458.734,E2 -7458.734} C_VEL
LIN {X 0,Y 467.752,Z 362.222,A -85,B 0,C 180,E1 -7462.228,E2 -7462.228} C_VEL
LIN {X 0,Y 467.726,Z 362.223,A -85,B 0,C 180,E1 -7464.828,E2 -7464.828} C_VEL
LIN {X 0,Y 467.863,Z 362.208,A -85,B 0,C 180,E1 -7467.417,E2 -7467.417} C_VEL
LIN {X 0,Y 467.887,Z 362.204,A -85,B 0,C 180,E1 -7470,E2 -7470} C_VEL
LIN {X 0,Y 467.862,Z 362.204,A -85,B 0,C 180,E1 -7472.583,E2 -7472.583} C_VEL
LIN {X 0,Y 467.739,Z 362.221,A -85,B 0,C 180,E1 -7476.038,E2 -7476.038} C_VEL
LIN {X 0,Y 467.685,Z 362.229,A -85,B 0,C 180,E1 -7478.643,E2 -7478.643} C_VEL
LIN {X 0,Y 467.66,Z 362.233,A -85,B 0,C 180,E1 -7482.146,E2 -7482.146} C_VEL
LIN {X 0,Y 467.643,Z 362.235,A -85,B 0,C 180,E1 -7485.695,E2 -7485.695} C_VEL
LIN {X 0,Y 467.621,Z 362.237,A -85,B 0,C 180,E1 -7488.765,E2 -7488.765} C_VEL
LIN {X 0,Y 467.584,Z 362.24,A -85,B 0,C 180,E1 -7491.268,E2 -7491.268} C_VEL
LIN {X 0,Y 467.567,Z 362.244,A -85,B 0,C 180,E1 -7493.944,E2 -7493.944} C_VEL
LIN {X 0,Y 467.616,Z 362.236,A -85,B 0,C 180,E1 -7496.801,E2 -7496.801} C_VEL
LIN {X 0,Y 467.558,Z 362.244,A -85,B 0,C 180,E1 -7499.738,E2 -7499.738} C_VEL
LIN {X 0,Y 467.587,Z 362.24,A -85,B 0,C 180,E1 -7502.758,E2 -7502.758} C_VEL
LIN {X 0,Y 467.557,Z 362.243,A -85,B 0,C 180,E1 -7505.89,E2 -7505.89} C_VEL
LIN {X 0,Y 467.585,Z 362.242,A -85,B 0,C 180,E1 -7509.145,E2 -7509.145} C_VEL
LIN {X 0,Y 467.589,Z 362.241,A -85,B 0,C 180,E1 -7512.567,E2 -7512.567} C_VEL
LIN {X 0,Y 467.569,Z 362.243,A -85,B 0,C 180,E1 -7515.053,E2 -7515.053} C_VEL
LIN {X 0,Y 467.592,Z 362.24,A -85,B 0,C 180,E1 -7517.44,E2 -7517.44} C_VEL
LIN {X 0,Y 467.586,Z 362.242,A -85,B 0,C 180,E1 -7520.855,E2 -7520.855} C_VEL
LIN {X 0,Y 467.566,Z 362.244,A -85,B 0,C 180,E1 -7524.26,E2 -7524.26} C_VEL
LIN {X 0,Y 467.585,Z 362.242,A -85,B 0,C 180,E1 -7527.321,E2 -7527.321} C_VEL
LIN {X 0,Y 467.704,Z 362.341,A -85,B 0,C 180,E1 -7529.651,E2 -7529.651} C_VEL
LIN {X 0,Y 467.597,Z 367.974,A -85,B 0,C 180,E1 -7532.471,E2 -7532.471} C_VEL
LIN {X 0,Y 467.408,Z 373.333,A -85,B 0,C 180,E1 -7535.101,E2 -7535.101} C_VEL
LIN {X 0,Y 467.267,Z 379.067,A -85,B 0,C 180,E1 -7537.913,E2 -7537.913} C_VEL
LIN {X 0,Y 467.192,Z 386.298,A -85,B 0,C 180,E1 -7541.391,E2 -7541.391} C_VEL
LIN {X 0,Y 467.11,Z 392.563,A -85,B 0,C 180,E1 -7544.351,E2 -7544.351} C_VEL
LIN {X 0,Y 466.958,Z 400.458,A -85,B 0,C 180,E1 -7548.041,E2 -7548.041} C_VEL
LIN {X 0,Y 466.869,Z 406.705,A -85,B 0,C 180,E1 -7550.824,E2 -7550.824} C_VEL
LIN {X 0,Y 468.169,Z 415.883,A -85,B 0,C 180,E1 -7551.258,E2 -7551.258} C_VEL
LIN {X 0,Y 468.055,Z 424.842,A -85,B 0,C 180,E1 -7551.799,E2 -7551.799} C_VEL
LIN {X 0,Y 467.824,Z 433.891,A -85,B 0,C 180,E1 -7552.527,E2 -7552.527} C_VEL
LIN {X 0,Y 467.49,Z 441.417,A -85,B 0,C 180,E1 -7553.309,E2 -7553.309} C_VEL
LIN {X 0,Y 467.47,Z 447.936,A -85,B 0,C 180,E1 -7554.176,E2 -7554.176} C_VEL
LIN {X 0,Y 467.336,Z 454.213,A -85,B 0,C 180,E1 -7555.256,E2 -7555.256} C_VEL
LIN {X 0,Y 467.199,Z 458.074,A -85,B 0,C 180,E1 -7556.118,E2 -7556.118} C_VEL
LIN {X 0,Y 467.105,Z 461.072,A -85,B 0,C 180,E1 -7556.981,E2 -7556.981} C_VEL
LIN {X 0,Y 466.901,Z 462.289,A -85,B 0,C 180,E1 -7557.412,E2 -7557.412} C_VEL
LIN {X 0,Y 466.795,Z 464.143,A -85,B 0,C 180,E1 -7558.274,E2 -7558.274} C_VEL
LIN {X 0,Y 466.772,Z 465.291,A -85,B 0,C 180,E1 -7559.137,E2 -7559.137} C_VEL
LIN {X 0,Y 466.774,Z 465.767,A -85,B 0,C 180,E1 -7560,E2 -7560} C_VEL
LIN {X 0,Y 466.791,Z 465.578,A -85,B 0,C 180,E1 -7560.863,E2 -7560.863} C_VEL
LIN {X 0,Y 466.834,Z 464.721,A -85,B 0,C 180,E1 -7561.725,E2 -7561.725} C_VEL
LIN {X 0,Y 466.932,Z 463.179,A -85,B 0,C 180,E1 -7562.588,E2 -7562.588} C_VEL
LIN {X 0,Y 467.121,Z 460.902,A -85,B 0,C 180,E1 -7563.45,E2 -7563.45} C_VEL
LIN {X 0,Y 467.284,Z 457.838,A -85,B 0,C 180,E1 -7564.313,E2 -7564.313} C_VEL
LIN {X 0,Y 467.563,Z 452.756,A -85,B 0,C 180,E1 -7565.391,E2 -7565.391} C_VEL
LIN {X 0,Y 467.63,Z 447.498,A -85,B 0,C 180,E1 -7566.255,E2 -7566.255} C_VEL
LIN {X 0,Y 467.918,Z 440.839,A -85,B 0,C 180,E1 -7567.116,E2 -7567.116} C_VEL
LIN {X 0,Y 468.246,Z 432.472,A -85,B 0,C 180,E1 -7567.959,E2 -7567.959} C_VEL
LIN {X 0,Y 468.467,Z 423.813,A -85,B 0,C 180,E1 -7568.628,E2 -7568.628} C_VEL
LIN {X 0,Y 468.423,Z 415.655,A -85,B 0,C 180,E1 -7569.118,E2 -7569.118} C_VEL
LIN {X 0,Y 467.067,Z 408.319,A -85,B 0,C 180,E1 -7569.5,E2 -7569.5} C_VEL
LIN {X 0,Y 467.224,Z 402.834,A -85,B 0,C 180,E1 -7572.157,E2 -7572.157} C_VEL
LIN {X 0,Y 467.385,Z 395.499,A -85,B 0,C 180,E1 -7575.769,E2 -7575.769} C_VEL
LIN {X 0,Y 467.563,Z 389.599,A -85,B 0,C 180,E1 -7578.744,E2 -7578.744} C_VEL
LIN {X 0,Y 467.753,Z 383.134,A -85,B 0,C 180,E1 -7582.063,E2 -7582.063} C_VEL
LIN {X 0,Y 468.005,Z 377.797,A -85,B 0,C 180,E1 -7584.865,E2 -7584.865} C_VEL
LIN {X 0,Y 468.281,Z 372.505,A -85,B 0,C 180,E1 -7587.727,E2 -7587.727} C_VEL
LIN {X 0,Y 468.462,Z 369.034,A -85,B 0,C 180,E1 -7589.675,E2 -7589.675} C_VEL
LIN {X 0,Y 468.171,Z 365.651,A -85,B 0,C 180,E1 -7591.696,E2 -7591.696} C_VEL
LIN {X 0,Y 467.599,Z 362.243,A -85,B 0,C 180,E1 -7594.014,E2 -7594.014} C_VEL
LIN {X 0,Y 467.553,Z 362.247,A -85,B 0,C 180,E1 -7597.187,E2 -7597.187} C_VEL
LIN {X 0,Y 467.601,Z 362.241,A -85,B 0,C 180,E1 -7600.262,E2 -7600.262} C_VEL
LIN {X 0,Y 467.622,Z 362.239,A -85,B 0,C 180,E1 -7602.571,E2 -7602.571} C_VEL
LIN {X 0,Y 467.57,Z 362.245,A -85,B 0,C 180,E1 -7606.177,E2 -7606.177} C_VEL
LIN {X 0,Y 467.585,Z 362.244,A -85,B 0,C 180,E1 -7608.723,E2 -7608.723} C_VEL
LIN {X 0,Y 467.568,Z 362.246,A -85,B 0,C 180,E1 -7611.955,E2 -7611.955} C_VEL
LIN {X 0,Y 467.611,Z 362.388,A -85,B 0,C 180,E1 -7614.455,E2 -7614.455} C_VEL
LIN {X 0,Y 469.165,Z 368.583,A -85,B 0,C 180,E1 -7617.021,E2 -7617.021} C_VEL
LIN {X 0,Y 471.052,Z 377.341,A -85,B 0,C 180,E1 -7619.923,E2 -7619.923} C_VEL
LIN {X 0,Y 471.584,Z 381.096,A -85,B 0,C 180,E1 -7621.03,E2 -7621.03} C_VEL
LIN {X 0,Y 471.113,Z 386.654,A -85,B 0,C 180,E1 -7622.454,E2 -7622.454} C_VEL
LIN {X 0,Y 469.718,Z 401.265,A -85,B 0,C 180,E1 -7625.88,E2 -7625.88} C_VEL
LIN {X 0,Y 468.687,Z 417.323,A -85,B 0,C 180,E1 -7629.367,E2 -7629.367} C_VEL
LIN {X 0,Y 468.009,Z 432.694,A -85,B 0,C 180,E1 -7632.522,E2 -7632.522} C_VEL
LIN {X 0,Y 467.64,Z 444.922,A -85,B 0,C 180,E1 -7634.947,E2 -7634.947} C_VEL
LIN {X 0,Y 469.131,Z 459.981,A -85,B 0,C 180,E1 -7635.37,E2 -7635.37} C_VEL
LIN {X 0,Y 469.367,Z 465.147,A -85,B 0,C 180,E1 -7635.558,E2 -7635.558} C_VEL
LIN {X 0,Y 469.016,Z 477.937,A -85,B 0,C 180,E1 -7636.128,E2 -7636.128} C_VEL
LIN {X 0,Y 468.597,Z 490.459,A -85,B 0,C 180,E1 -7636.888,E2 -7636.888} C_VEL
LIN {X 0,Y 468.263,Z 501.364,A -85,B 0,C 180,E1 -7637.733,E2 -7637.733} C_VEL
LIN {X 0,Y 467.785,Z 511.718,A -85,B 0,C 180,E1 -7638.737,E2 -7638.737} C_VEL
LIN {X 0,Y 467.413,Z 520.839,A -85,B 0,C 180,E1 -7639.824,E2 -7639.824} C_VEL
LIN {X 0,Y 467.112,Z 529.72,A -85,B 0,C 180,E1 -7641.128,E2 -7641.128} C_VEL
LIN {X 0,Y 466.949,Z 536.789,A -85,B 0,C 180,E1 -7642.432,E2 -7642.432} C_VEL
LIN {X 0,Y 466.835,Z 543.271,A -85,B 0,C 180,E1 -7643.951,E2 -7643.951} C_VEL
LIN {X 0,Y 466.742,Z 547.48,A -85,B 0,C 180,E1 -7645.249,E2 -7645.249} C_VEL
LIN {X 0,Y 466.82,Z 550.597,A -85,B 0,C 180,E1 -7646.547,E2 -7646.547} C_VEL
LIN {X 0,Y 466.818,Z 552.097,A -85,B 0,C 180,E1 -7647.411,E2 -7647.411} C_VEL
LIN {X 0,Y 466.673,Z 553.805,A -85,B 0,C 180,E1 -7649.137,E2 -7649.137} C_VEL
LIN {X 0,Y 466.673,Z 554.055,A -85,B 0,C 180,E1 -7650,E2 -7650} C_VEL
LIN {X 0,Y 466.669,Z 553.849,A -85,B 0,C 180,E1 -7650.863,E2 -7650.863} C_VEL
LIN {X 0,Y 466.818,Z 552.243,A -85,B 0,C 180,E1 -7652.589,E2 -7652.589} C_VEL
LIN {X 0,Y 466.817,Z 550.782,A -85,B 0,C 180,E1 -7653.452,E2 -7653.452} C_VEL
LIN {X 0,Y 466.729,Z 547.735,A -85,B 0,C 180,E1 -7654.75,E2 -7654.75} C_VEL
LIN {X 0,Y 466.809,Z 543.602,A -85,B 0,C 180,E1 -7656.049,E2 -7656.049} C_VEL
LIN {X 0,Y 466.949,Z 537.232,A -85,B 0,C 180,E1 -7657.567,E2 -7657.567} C_VEL
LIN {X 0,Y 467.112,Z 530.258,A -85,B 0,C 180,E1 -7658.871,E2 -7658.871} C_VEL
LIN {X 0,Y 467.414,Z 521.472,A -85,B 0,C 180,E1 -7660.176,E2 -7660.176} C_VEL
LIN {X 0,Y 467.836,Z 511.458,A -85,B 0,C 180,E1 -7661.371,E2 -7661.371} C_VEL
LIN {X 0,Y 468.277,Z 500.472,A -85,B 0,C 180,E1 -7662.411,E2 -7662.411} C_VEL
LIN {X 0,Y 468.682,Z 489.81,A -85,B 0,C 180,E1 -7663.219,E2 -7663.219} C_VEL
LIN {X 0,Y 469.08,Z 477.943,A -85,B 0,C 180,E1 -7663.925,E2 -7663.925} C_VEL
LIN {X 0,Y 469.454,Z 464.801,A -85,B 0,C 180,E1 -7664.494,E2 -7664.494} C_VEL
LIN {X 0,Y 469.205,Z 460.29,A -85,B 0,C 180,E1 -7664.655,E2 -7664.655} C_VEL
LIN {X 0,Y 467.912,Z 447.722,A -85,B 0,C 180,E1 -7665.002,E2 -7665.002} C_VEL
LIN {X 0,Y 467.683,Z 445.452,A -85,B 0,C 180,E1 -7665.079,E2 -7665.079} C_VEL
LIN {X 0,Y 468.23,Z 429.056,A -85,B 0,C 180,E1 -7668.373,E2 -7668.373} C_VEL
LIN {X 0,Y 468.954,Z 414.207,A -85,B 0,C 180,E1 -7671.403,E2 -7671.403} C_VEL
LIN {X 0,Y 469.765,Z 400,A -85,B 0,C 180,E1 -7674.375,E2 -7674.375} C_VEL
LIN {X 0,Y 470.916,Z 383.294,A -85,B 0,C 180,E1 -7677.944,E2 -7677.944} C_VEL
LIN {X 0,Y 471.039,Z 378.515,A -85,B 0,C 180,E1 -7679.006,E2 -7679.006} C_VEL
LIN {X 0,Y 468.495,Z 366.503,A -85,B 0,C 180,E1 -7681.919,E2 -7681.919} C_VEL
LIN {X 0,Y 467.599,Z 362.241,A -85,B 0,C 180,E1 -7683.013,E2 -7683.013} C_VEL
LIN {X 0,Y 467.555,Z 362.244,A -85,B 0,C 180,E1 -7685.889,E2 -7685.889} C_VEL
LIN {X 0,Y 467.583,Z 362.239,A -85,B 0,C 180,E1 -7689.145,E2 -7689.145} C_VEL
LIN {X 0,Y 467.587,Z 362.24,A -85,B 0,C 180,E1 -7692.567,E2 -7692.567} C_VEL
LIN {X 0,Y 467.572,Z 362.243,A -85,B 0,C 180,E1 -7695.053,E2 -7695.053} C_VEL
LIN {X 0,Y 467.59,Z 362.24,A -85,B 0,C 180,E1 -7697.44,E2 -7697.44} C_VEL
LIN {X 0,Y 467.584,Z 362.239,A -85,B 0,C 180,E1 -7700.855,E2 -7700.855} C_VEL
LIN {X 0,Y 467.564,Z 362.243,A -85,B 0,C 180,E1 -7704.26,E2 -7704.26} C_VEL
LIN {X 0,Y 467.583,Z 362.242,A -85,B 0,C 180,E1 -7707.321,E2 -7707.321} C_VEL
LIN {X 0,Y 467.571,Z 362.241,A -85,B 0,C 180,E1 -7710.667,E2 -7710.667} C_VEL
LIN {X 0,Y 467.618,Z 362.236,A -85,B 0,C 180,E1 -7713.2,E2 -7713.2} C_VEL
LIN {X 0,Y 467.593,Z 362.241,A -85,B 0,C 180,E1 -7716.468,E2 -7716.468} C_VEL
LIN {X 0,Y 467.625,Z 362.236,A -85,B 0,C 180,E1 -7719.777,E2 -7719.777} C_VEL
LIN {X 0,Y 467.61,Z 362.235,A -85,B 0,C 180,E1 -7722.507,E2 -7722.507} C_VEL
LIN {X 0,Y 467.611,Z 362.239,A -85,B 0,C 180,E1 -7725.197,E2 -7725.197} C_VEL
LIN {X 0,Y 467.657,Z 362.232,A -85,B 0,C 180,E1 -7727.855,E2 -7727.855} C_VEL
LIN {X 0,Y 467.683,Z 362.228,A -85,B 0,C 180,E1 -7731.357,E2 -7731.357} C_VEL
LIN {X 0,Y 467.745,Z 362.22,A -85,B 0,C 180,E1 -7733.963,E2 -7733.963} C_VEL
LIN {X 0,Y 467.861,Z 362.207,A -85,B 0,C 180,E1 -7737.417,E2 -7737.417} C_VEL
LIN {X 0,Y 467.885,Z 362.206,A -85,B 0,C 180,E1 -7740,E2 -7740} C_VEL
LIN {X 0,Y 467.861,Z 362.205,A -85,B 0,C 180,E1 -7742.583,E2 -7742.583} C_VEL
LIN {X 0,Y 467.745,Z 362.219,A -85,B 0,C 180,E1 -7746.037,E2 -7746.037} C_VEL
LIN {X 0,Y 467.684,Z 362.23,A -85,B 0,C 180,E1 -7748.643,E2 -7748.643} C_VEL
LIN {X 0,Y 467.685,Z 362.229,A -85,B 0,C 180,E1 -7752.145,E2 -7752.145} C_VEL
LIN {X 0,Y 467.651,Z 362.23,A -85,B 0,C 180,E1 -7755.885,E2 -7755.885} C_VEL
LIN {X 0,Y 467.626,Z 362.235,A -85,B 0,C 180,E1 -7759.308,E2 -7759.308} C_VEL
LIN {X 0,Y 467.538,Z 362.247,A -85,B 0,C 180,E1 -7762.074,E2 -7762.074} C_VEL
LIN {X 0,Y 467.605,Z 362.238,A -85,B 0,C 180,E1 -7764.887,E2 -7764.887} C_VEL
LIN {X 0,Y 467.621,Z 362.234,A -85,B 0,C 180,E1 -7767.769,E2 -7767.769} C_VEL
LIN {X 0,Y 467.57,Z 362.242,A -85,B 0,C 180,E1 -7771.045,E2 -7771.045} C_VEL
LIN {X 0,Y 467.591,Z 362.24,A -85,B 0,C 180,E1 -7774.243,E2 -7774.243} C_VEL
LIN {X 0,Y 467.551,Z 362.245,A -85,B 0,C 180,E1 -7777.187,E2 -7777.187} C_VEL
LIN {X 0,Y 467.579,Z 362.243,A -85,B 0,C 180,E1 -7780.265,E2 -7780.265} C_VEL
LIN {X 0,Y 467.588,Z 362.241,A -85,B 0,C 180,E1 -7782.567,E2 -7782.567} C_VEL
LIN {X 0,Y 467.572,Z 362.245,A -85,B 0,C 180,E1 -7785.053,E2 -7785.053} C_VEL
LIN {X 0,Y 467.59,Z 362.239,A -85,B 0,C 180,E1 -7787.44,E2 -7787.44} C_VEL
LIN {X 0,Y 467.584,Z 362.241,A -85,B 0,C 180,E1 -7790.856,E2 -7790.856} C_VEL
LIN {X 0,Y 467.561,Z 362.244,A -85,B 0,C 180,E1 -7794.261,E2 -7794.261} C_VEL
LIN {X 0,Y 467.584,Z 362.24,A -85,B 0,C 180,E1 -7797.321,E2 -7797.321} C_VEL
LIN {X 0,Y 467.572,Z 362.243,A -85,B 0,C 180,E1 -7800.667,E2 -7800.667} C_VEL
LIN {X 0,Y 467.619,Z 362.237,A -85,B 0,C 180,E1 -7803.2,E2 -7803.2} C_VEL
LIN {X 0,Y 467.595,Z 362.24,A -85,B 0,C 180,E1 -7806.468,E2 -7806.468} C_VEL
LIN {X 0,Y 467.627,Z 362.234,A -85,B 0,C 180,E1 -7809.778,E2 -7809.778} C_VEL
LIN {X 0,Y 467.612,Z 362.237,A -85,B 0,C 180,E1 -7812.507,E2 -7812.507} C_VEL
LIN {X 0,Y 467.61,Z 362.238,A -85,B 0,C 180,E1 -7815.197,E2 -7815.197} C_VEL
LIN {X 0,Y 467.6,Z 362.238,A -85,B 0,C 180,E1 -7815.421,E2 -7815.421} C_VEL
LIN {X 0,Y 466.93,Z 362.323,A -85,B 0,C 180,E1 -7816.14,E2 -7816.14} C_VEL
LIN {X 0,Y 464.086,Z 362.677,A -85,B 0,C 180,E1 -7817.309,E2 -7817.309} C_VEL
LIN {X 0,Y 461.688,Z 362.976,A -85,B 0,C 180,E1 -7818.251,E2 -7818.251} C_VEL
LIN {X 0,Y 460.661,Z 363.103,A -85,B 0,C 180,E1 -7818.978,E2 -7818.978} C_VEL
LIN {X 0,Y 460.58,Z 363.112,A -85,B 0,C 180,E1 -7819.225,E2 -7819.225} C_VEL
LIN {X 0,Y 460.718,Z 363.095,A -85,B 0,C 180,E1 -7822.543,E2 -7822.543} C_VEL
LIN {X 0,Y 460.698,Z 363.098,A -85,B 0,C 180,E1 -7824.748,E2 -7824.748} C_VEL
LIN {X 0,Y 460.803,Z 363.087,A -85,B 0,C 180,E1 -7827.378,E2 -7827.378} C_VEL
